LIN {X 0,Y 383.012,Z 410.276,A -85,B 0,C 180,E1 -11840.414,E2 -11840.414} C_VEL
LIN {X 0,Y 383.022,Z 410.276,A -85,B 0,C 180,E1 -11844.045,E2 -11844.045} C_VEL
LIN {X 0,Y 383.032,Z 410.273,A -85,B 0,C 180,E1 -11847.853,E2 -11847.853} C_VEL
LIN {X 0,Y 383.059,Z 410.269,A -85,B 0,C 180,E1 -11851.721,E2 -11851.721} C_VEL
LIN {X 0,Y 383.047,Z 410.267,A -85,B 0,C 180,E1 -11855.04,E2 -11855.04} C_VEL
LIN {X 0,Y 382.989,Z 410.276,A -85,B 0,C 180,E1 -11858.469,E2 -11858.469} C_VEL
LIN {X 0,Y 383.085,Z 410.269,A -85,B 0,C 180,E1 -11861.828,E2 -11861.828} C_VEL
LIN {X 0,Y 383.108,Z 410.26,A -85,B 0,C 180,E1 -11865.119,E2 -11865.119} C_VEL
LIN {X 0,Y 383.093,Z 410.263,A -85,B 0,C 180,E1 -11868.358,E2 -11868.358} C_VEL
LIN {X 0,Y 383.3,Z 410.24,A -85,B 0,C 180,E1 -11871.934,E2 -11871.934} C_VEL
LIN {X 0,Y 383.196,Z 410.249,A -85,B 0,C 180,E1 -11874.739,E2 -11874.739} C_VEL
LIN {X 0,Y 383.384,Z 410.229,A -85,B 0,C 180,E1 -11877.899,E2 -11877.899} C_VEL
LIN {X 0,Y 383.516,Z 410.211,A -85,B 0,C 180,E1 -11880.001,E2 -11880.001} C_VEL
LIN {X 0,Y 383.249,Z 410.245,A -85,B 0,C 180,E1 -11883.154,E2 -11883.154} C_VEL
LIN {X 0,Y 383.284,Z 410.238,A -85,B 0,C 180,E1 -11886.317,E2 -11886.317} C_VEL
LIN {X 0,Y 383.257,Z 410.241,A -85,B 0,C 180,E1 -11888.436,E2 -11888.436} C_VEL
LIN {X 0,Y 383.095,Z 410.266,A -85,B 0,C 180,E1 -11891.643,E2 -11891.643} C_VEL
LIN {X 0,Y 383.108,Z 410.261,A -85,B 0,C 180,E1 -11894.882,E2 -11894.882} C_VEL
LIN {X 0,Y 383.061,Z 410.266,A -85,B 0,C 180,E1 -11898.174,E2 -11898.174} C_VEL
LIN {X 0,Y 382.991,Z 410.278,A -85,B 0,C 180,E1 -11901.532,E2 -11901.532} C_VEL
LIN {X 0,Y 383.051,Z 410.271,A -85,B 0,C 180,E1 -11904.961,E2 -11904.961} C_VEL
LIN {X 0,Y 383.028,Z 410.27,A -85,B 0,C 180,E1 -11908.271,E2 -11908.271} C_VEL
LIN {X 0,Y 383.008,Z 410.272,A -85,B 0,C 180,E1 -11912.15,E2 -11912.15} C_VEL
LIN {X 0,Y 383.018,Z 410.274,A -85,B 0,C 180,E1 -11914.669,E2 -11914.669} C_VEL
LIN {X 0,Y 383.004,Z 410.278,A -85,B 0,C 180,E1 -11917.905,E2 -11917.905} C_VEL
LIN {X 0,Y 383.441,Z 413.021,A -85,B 0,C 180,E1 -11921.288,E2 -11921.288} C_VEL
LIN {X 0,Y 383.863,Z 416.004,A -85,B 0,C 180,E1 -11924.436,E2 -11924.436} C_VEL
LIN {X 0,Y 384.216,Z 419.062,A -85,B 0,C 180,E1 -11927.407,E2 -11927.407} C_VEL
LIN {X 0,Y 384.099,Z 422.233,A -85,B 0,C 180,E1 -11930.219,E2 -11930.219} C_VEL
LIN {X 0,Y 383.629,Z 426.471,A -85,B 0,C 180,E1 -11933.714,E2 -11933.714} C_VEL
LIN {X 0,Y 383.227,Z 430.206,A -85,B 0,C 180,E1 -11936.622,E2 -11936.622} C_VEL
LIN {X 0,Y 382.802,Z 435.145,A -85,B 0,C 180,E1 -11940.284,E2 -11940.284} C_VEL
LIN {X 0,Y 382.563,Z 438.484,A -85,B 0,C 180,E1 -11942.66,E2 -11942.66} C_VEL
LIN {X 0,Y 382.356,Z 441.851,A -85,B 0,C 180,E1 -11944.991,E2 -11944.991} C_VEL
LIN {X 0,Y 382.084,Z 446.961,A -85,B 0,C 180,E1 -11948.415,E2 -11948.415} C_VEL
LIN {X 0,Y 381.915,Z 451.227,A -85,B 0,C 180,E1 -11951.101,E2 -11951.101} C_VEL
LIN {X 0,Y 383.99,Z 461.506,A -85,B 0,C 180,E1 -11951.544,E2 -11951.544} C_VEL
LIN {X 0,Y 385.644,Z 470.976,A -85,B 0,C 180,E1 -11952.061,E2 -11952.061} C_VEL
LIN {X 0,Y 386.955,Z 479.684,A -85,B 0,C 180,E1 -11952.632,E2 -11952.632} C_VEL
LIN {X 0,Y 387.304,Z 485.306,A -85,B 0,C 180,E1 -11953.027,E2 -11953.027} C_VEL
LIN {X 0,Y 386.288,Z 497.459,A -85,B 0,C 180,E1 -11954.027,E2 -11954.027} C_VEL
LIN {X 0,Y 385.499,Z 506.412,A -85,B 0,C 180,E1 -11954.943,E2 -11954.943} C_VEL
LIN {X 0,Y 384.91,Z 513.425,A -85,B 0,C 180,E1 -11955.786,E2 -11955.786} C_VEL
LIN {X 0,Y 384.102,Z 522.165,A -85,B 0,C 180,E1 -11957.048,E2 -11957.048} C_VEL
LIN {X 0,Y 383.437,Z 528.368,A -85,B 0,C 180,E1 -11958.1,E2 -11958.1} C_VEL
LIN {X 0,Y 382.892,Z 534.91,A -85,B 0,C 180,E1 -11959.423,E2 -11959.423} C_VEL
LIN {X 0,Y 382.464,Z 539.413,A -85,B 0,C 180,E1 -11960.481,E2 -11960.481} C_VEL
LIN {X 0,Y 382.033,Z 544.907,A -85,B 0,C 180,E1 -11962.069,E2 -11962.069} C_VEL
LIN {X 0,Y 381.769,Z 549.234,A -85,B 0,C 180,E1 -11963.658,E2 -11963.658} C_VEL
LIN {X 0,Y 381.682,Z 551.602,A -85,B 0,C 180,E1 -11964.717,E2 -11964.717} C_VEL
LIN {X 0,Y 381.642,Z 553.402,A -85,B 0,C 180,E1 -11965.776,E2 -11965.776} C_VEL
LIN {X 0,Y 381.558,Z 555.847,A -85,B 0,C 180,E1 -11967.889,E2 -11967.889} C_VEL
LIN {X 0,Y 381.591,Z 556.437,A -85,B 0,C 180,E1 -11968.944,E2 -11968.944} C_VEL
LIN {X 0,Y 381.591,Z 556.437,A -85,B 0,C 180,E1 -11971.055,E2 -11971.055} C_VEL
LIN {X 0,Y 381.558,Z 555.848,A -85,B 0,C 180,E1 -11972.111,E2 -11972.111} C_VEL
LIN {X 0,Y 381.642,Z 553.403,A -85,B 0,C 180,E1 -11974.224,E2 -11974.224} C_VEL
LIN {X 0,Y 381.693,Z 550.488,A -85,B 0,C 180,E1 -11975.796,E2 -11975.796} C_VEL
LIN {X 0,Y 381.934,Z 546.463,A -85,B 0,C 180,E1 -11977.4,E2 -11977.4} C_VEL
LIN {X 0,Y 382.305,Z 541.331,A -85,B 0,C 180,E1 -11978.989,E2 -11978.989} C_VEL
LIN {X 0,Y 382.759,Z 536.068,A -85,B 0,C 180,E1 -11980.313,E2 -11980.313} C_VEL
LIN {X 0,Y 383.293,Z 529.747,A -85,B 0,C 180,E1 -11981.636,E2 -11981.636} C_VEL
LIN {X 0,Y 383.909,Z 523.795,A -85,B 0,C 180,E1 -11982.69,E2 -11982.69} C_VEL
LIN {X 0,Y 384.57,Z 516.865,A -85,B 0,C 180,E1 -11983.743,E2 -11983.743} C_VEL
LIN {X 0,Y 385.262,Z 508.68,A -85,B 0,C 180,E1 -11984.796,E2 -11984.796} C_VEL
LIN {X 0,Y 386.03,Z 500.167,A -85,B 0,C 180,E1 -11985.712,E2 -11985.712} C_VEL
LIN {X 0,Y 386.744,Z 491.448,A -85,B 0,C 180,E1 -11986.495,E2 -11986.495} C_VEL
LIN {X 0,Y 387.323,Z 482.508,A -85,B 0,C 180,E1 -11987.161,E2 -11987.161} C_VEL
LIN {X 0,Y 385.932,Z 472.449,A -85,B 0,C 180,E1 -11987.848,E2 -11987.848} C_VEL
LIN {X 0,Y 384.09,Z 461.865,A -85,B 0,C 180,E1 -11988.437,E2 -11988.437} C_VEL
LIN {X 0,Y 381.971,Z 451.872,A -85,B 0,C 180,E1 -11988.879,E2 -11988.879} C_VEL
LIN {X 0,Y 381.884,Z 451.048,A -85,B 0,C 180,E1 -11988.926,E2 -11988.926} C_VEL
LIN {X 0,Y 382.184,Z 445.234,A -85,B 0,C 180,E1 -11992.716,E2 -11992.716} C_VEL
LIN {X 0,Y 382.45,Z 440.161,A -85,B 0,C 180,E1 -11996.169,E2 -11996.169} C_VEL
LIN {X 0,Y 382.796,Z 435.146,A -85,B 0,C 180,E1 -11999.716,E2 -11999.716} C_VEL
LIN {X 0,Y 383.224,Z 430.206,A -85,B 0,C 180,E1 -12003.378,E2 -12003.378} C_VEL
LIN {X 0,Y 383.748,Z 425.351,A -85,B 0,C 180,E1 -12007.182,E2 -12007.182} C_VEL
LIN {X 0,Y 384.098,Z 422.187,A -85,B 0,C 180,E1 -12009.821,E2 -12009.821} C_VEL
LIN {X 0,Y 384.212,Z 419.044,A -85,B 0,C 180,E1 -12012.593,E2 -12012.593} C_VEL
LIN {X 0,Y 383.827,Z 415.64,A -85,B 0,C 180,E1 -12015.909,E2 -12015.909} C_VEL
LIN {X 0,Y 383.416,Z 412.995,A -85,B 0,C 180,E1 -12018.722,E2 -12018.722} C_VEL
LIN {X 0,Y 383.001,Z 410.279,A -85,B 0,C 180,E1 -12022.095,E2 -12022.095} C_VEL
LIN {X 0,Y 383.015,Z 410.277,A -85,B 0,C 180,E1 -12025.331,E2 -12025.331} C_VEL
LIN {X 0,Y 383.034,Z 410.269,A -85,B 0,C 180,E1 -12027.852,E2 -12027.852} C_VEL
LIN {X 0,Y 383.06,Z 410.266,A -85,B 0,C 180,E1 -12031.719,E2 -12031.719} C_VEL
LIN {X 0,Y 383.048,Z 410.271,A -85,B 0,C 180,E1 -12035.039,E2 -12035.039} C_VEL
LIN {X 0,Y 382.988,Z 410.278,A -85,B 0,C 180,E1 -12038.468,E2 -12038.468} C_VEL
LIN {X 0,Y 383.058,Z 410.266,A -85,B 0,C 180,E1 -12041.826,E2 -12041.826} C_VEL
LIN {X 0,Y 383.105,Z 410.262,A -85,B 0,C 180,E1 -12045.118,E2 -12045.118} C_VEL
LIN {X 0,Y 383.093,Z 410.266,A -85,B 0,C 180,E1 -12048.357,E2 -12048.357} C_VEL
LIN {X 0,Y 383.298,Z 410.237,A -85,B 0,C 180,E1 -12051.932,E2 -12051.932} C_VEL
LIN {X 0,Y 383.194,Z 410.253,A -85,B 0,C 180,E1 -12054.738,E2 -12054.738} C_VEL
LIN {X 0,Y 383.382,Z 410.227,A -85,B 0,C 180,E1 -12057.898,E2 -12057.898} C_VEL
LIN {X 0,Y 383.513,Z 410.212,A -85,B 0,C 180,E1 -12059.999,E2 -12059.999} C_VEL
LIN {X 0,Y 383.246,Z 410.243,A -85,B 0,C 180,E1 -12063.153,E2 -12063.153} C_VEL
LIN {X 0,Y 383.262,Z 410.243,A -85,B 0,C 180,E1 -12066.636,E2 -12066.636} C_VEL
LIN {X 0,Y 383.253,Z 410.246,A -85,B 0,C 180,E1 -12068.435,E2 -12068.435} C_VEL
LIN {X 0,Y 383.09,Z 410.263,A -85,B 0,C 180,E1 -12071.642,E2 -12071.642} C_VEL
LIN {X 0,Y 383.106,Z 410.26,A -85,B 0,C 180,E1 -12074.881,E2 -12074.881} C_VEL
LIN {X 0,Y 383.082,Z 410.269,A -85,B 0,C 180,E1 -12078.172,E2 -12078.172} C_VEL
LIN {X 0,Y 382.986,Z 410.276,A -85,B 0,C 180,E1 -12081.531,E2 -12081.531} C_VEL
LIN {X 0,Y 383.045,Z 410.267,A -85,B 0,C 180,E1 -12084.96,E2 -12084.96} C_VEL
LIN {X 0,Y 383.042,Z 410.269,A -85,B 0,C 180,E1 -12088.492,E2 -12088.492} C_VEL
LIN {X 0,Y 383.001,Z 410.274,A -85,B 0,C 180,E1 -12092.427,E2 -12092.427} C_VEL
LIN {X 0,Y 383.027,Z 410.273,A -85,B 0,C 180,E1 -12096.165,E2 -12096.165} C_VEL
LIN {X 0,Y 383.014,Z 410.276,A -85,B 0,C 180,E1 -12099.957,E2 -12099.957} C_VEL
LIN {X 0,Y 383.059,Z 410.266,A -85,B 0,C 180,E1 -12102.788,E2 -12102.788} C_VEL
LIN {X 0,Y 383.063,Z 410.271,A -85,B 0,C 180,E1 -12105.8,E2 -12105.8} C_VEL
LIN {X 0,Y 383.038,Z 410.269,A -85,B 0,C 180,E1 -12108.786,E2 -12108.786} C_VEL
LIN {X 0,Y 382.997,Z 410.275,A -85,B 0,C 180,E1 -12112.096,E2 -12112.096} C_VEL
LIN {X 0,Y 383.012,Z 410.276,A -85,B 0,C 180,E1 -12115.332,E2 -12115.332} C_VEL
LIN {X 0,Y 382.977,Z 410.278,A -85,B 0,C 180,E1 -12119.082,E2 -12119.082} C_VEL
LIN {X 0,Y 383.051,Z 410.267,A -85,B 0,C 180,E1 -12122.698,E2 -12122.698} C_VEL
LIN {X 0,Y 383.029,Z 410.27,A -85,B 0,C 180,E1 -12126.193,E2 -12126.193} C_VEL
LIN {X 0,Y 383.05,Z 410.272,A -85,B 0,C 180,E1 -12129.599,E2 -12129.599} C_VEL
LIN {X 0,Y 383.1,Z 410.267,A -85,B 0,C 180,E1 -12132.932,E2 -12132.932} C_VEL
LIN {X 0,Y 383.121,Z 410.263,A -85,B 0,C 180,E1 -12136.464,E2 -12136.464} C_VEL
LIN {X 0,Y 383.138,Z 410.29,A -85,B 0,C 180,E1 -12139.598,E2 -12139.598} C_VEL
LIN {X 0,Y 383.821,Z 412.514,A -85,B 0,C 180,E1 -12139.95,E2 -12139.95} C_VEL
LIN {X 0,Y 385.2,Z 414.425,A -85,B 0,C 180,E1 -12140.616,E2 -12140.616} C_VEL
LIN {X 0,Y 387.436,Z 415.861,A -85,B 0,C 180,E1 -12141.656,E2 -12141.656} C_VEL
LIN {X 0,Y 388.84,Z 416.571,A -85,B 0,C 180,E1 -12142.402,E2 -12142.402} C_VEL
LIN {X 0,Y 389.961,Z 418.835,A -85,B 0,C 180,E1 -12143.142,E2 -12143.142} C_VEL
LIN {X 0,Y 391.789,Z 420.996,A -85,B 0,C 180,E1 -12144.467,E2 -12144.467} C_VEL
LIN {X 0,Y 393.422,Z 422.061,A -85,B 0,C 180,E1 -12145.903,E2 -12145.903} C_VEL
LIN {X 0,Y 394.945,Z 422.431,A -85,B 0,C 180,E1 -12147.961,E2 -12147.961} C_VEL
LIN {X 0,Y 395.509,Z 422.495,A -85,B 0,C 180,E1 -12150,E2 -12150} C_VEL
LIN {X 0,Y 394.944,Z 422.431,A -85,B 0,C 180,E1 -12152.04,E2 -12152.04} C_VEL
LIN {X 0,Y 393.422,Z 422.061,A -85,B 0,C 180,E1 -12154.098,E2 -12154.098} C_VEL
LIN {X 0,Y 391.445,Z 420.7,A -85,B 0,C 180,E1 -12155.796,E2 -12155.796} C_VEL
LIN {X 0,Y 389.551,Z 418.154,A -85,B 0,C 180,E1 -12157.135,E2 -12157.135} C_VEL
LIN {X 0,Y 388.788,Z 416.393,A -85,B 0,C 180,E1 -12157.634,E2 -12157.634} C_VEL
LIN {X 0,Y 385.957,Z 415.054,A -85,B 0,C 180,E1 -12159.036,E2 -12159.036} C_VEL
LIN {X 0,Y 384.054,Z 412.961,A -85,B 0,C 180,E1 -12159.938,E2 -12159.938} C_VEL
LIN {X 0,Y 383.253,Z 410.919,A -85,B 0,C 180,E1 -12160.333,E2 -12160.333} C_VEL
LIN {X 0,Y 383.122,Z 410.263,A -85,B 0,C 180,E1 -12160.437,E2 -12160.437} C_VEL
LIN {X 0,Y 383.123,Z 410.262,A -85,B 0,C 180,E1 -12163.796,E2 -12163.796} C_VEL
LIN {X 0,Y 383.091,Z 410.267,A -85,B 0,C 180,E1 -12167.455,E2 -12167.455} C_VEL
LIN {X 0,Y 383.025,Z 410.276,A -85,B 0,C 180,E1 -12170.647,E2 -12170.647} C_VEL
LIN {X 0,Y 383.03,Z 410.27,A -85,B 0,C 180,E1 -12173.807,E2 -12173.807} C_VEL
LIN {X 0,Y 383.053,Z 410.267,A -85,B 0,C 180,E1 -12177.302,E2 -12177.302} C_VEL
LIN {X 0,Y 382.978,Z 410.278,A -85,B 0,C 180,E1 -12180.919,E2 -12180.919} C_VEL
LIN {X 0,Y 383.014,Z 410.276,A -85,B 0,C 180,E1 -12184.668,E2 -12184.668} C_VEL
LIN {X 0,Y 382.995,Z 410.274,A -85,B 0,C 180,E1 -12185.381,E2 -12185.381} C_VEL
LIN {X 0,Y 382.352,Z 410.358,A -85,B 0,C 180,E1 -12186.258,E2 -12186.258} C_VEL
LIN {X 0,Y 379.535,Z 410.71,A -85,B 0,C 180,E1 -12187.686,E2 -12187.686} C_VEL
LIN {X 0,Y 377.13,Z 411.01,A -85,B 0,C 180,E1 -12188.841,E2 -12188.841} C_VEL
LIN {X 0,Y 376.084,Z 411.138,A -85,B 0,C 180,E1 -12189.733,E2 -12189.733} C_VEL
LIN {X 0,Y 375.992,Z 411.148,A -85,B 0,C 180,E1 -12190.035,E2 -12190.035} C_VEL
LIN {X 0,Y 375.984,Z 411.147,A -85,B 0,C 180,E1 -12193.198,E2 -12193.198} C_VEL
LIN {X 0,Y 375.932,Z 411.155,A -85,B 0,C 180,E1 -12196.81,E2 -12196.81} C_VEL
LIN {X 0,Y 375.959,Z 411.153,A -85,B 0,C 180,E1 -12200.538,E2 -12200.538} C_VEL
LIN {X 0,Y 375.96,Z 411.151,A -85,B 0,C 180,E1 -12203.496,E2 -12203.496} C_VEL
LIN {X 0,Y 375.959,Z 411.154,A -85,B 0,C 180,E1 -12205.889,E2 -12205.889} C_VEL
LIN {X 0,Y 375.965,Z 411.152,A -85,B 0,C 180,E1 -12209.688,E2 -12209.688} C_VEL
LIN {X 0,Y 375.998,Z 411.151,A -85,B 0,C 180,E1 -12212.142,E2 -12212.142} C_VEL
LIN {X 0,Y 376.001,Z 411.146,A -85,B 0,C 180,E1 -12214.539,E2 -12214.539} C_VEL
LIN {X 0,Y 375.959,Z 411.156,A -85,B 0,C 180,E1 -12218.046,E2 -12218.046} C_VEL
LIN {X 0,Y 376.02,Z 411.145,A -85,B 0,C 180,E1 -12221.474,E2 -12221.474} C_VEL
LIN {X 0,Y 376.057,Z 411.138,A -85,B 0,C 180,E1 -12224.833,E2 -12224.833} C_VEL
LIN {X 0,Y 376.046,Z 411.142,A -85,B 0,C 180,E1 -12228.137,E2 -12228.137} C_VEL
LIN {X 0,Y 376.254,Z 411.119,A -85,B 0,C 180,E1 -12231.878,E2 -12231.878} C_VEL
LIN {X 0,Y 376.168,Z 411.124,A -85,B 0,C 180,E1 -12234.64,E2 -12234.64} C_VEL
LIN {X 0,Y 376.35,Z 411.106,A -85,B 0,C 180,E1 -12237.86,E2 -12237.86} C_VEL
LIN {X 0,Y 376.485,Z 411.087,A -85,B 0,C 180,E1 -12240.001,E2 -12240.001} C_VEL
LIN {X 0,Y 376.187,Z 411.125,A -85,B 0,C 180,E1 -12243.214,E2 -12243.214} C_VEL
LIN {X 0,Y 376.244,Z 411.115,A -85,B 0,C 180,E1 -12246.436,E2 -12246.436} C_VEL
LIN {X 0,Y 376.203,Z 411.12,A -85,B 0,C 180,E1 -12248.596,E2 -12248.596} C_VEL
LIN {X 0,Y 376.048,Z 411.141,A -85,B 0,C 180,E1 -12251.864,E2 -12251.864} C_VEL
LIN {X 0,Y 376.056,Z 411.142,A -85,B 0,C 180,E1 -12255.168,E2 -12255.168} C_VEL
LIN {X 0,Y 376.007,Z 411.144,A -85,B 0,C 180,E1 -12258.527,E2 -12258.527} C_VEL
LIN {X 0,Y 375.961,Z 411.151,A -85,B 0,C 180,E1 -12261.955,E2 -12261.955} C_VEL
LIN {X 0,Y 376.005,Z 411.148,A -85,B 0,C 180,E1 -12265.462,E2 -12265.462} C_VEL
LIN {X 0,Y 375.96,Z 411.156,A -85,B 0,C 180,E1 -12269.081,E2 -12269.081} C_VEL
LIN {X 0,Y 375.948,Z 411.155,A -85,B 0,C 180,E1 -12272.829,E2 -12272.829} C_VEL
LIN {X 0,Y 375.958,Z 411.157,A -85,B 0,C 180,E1 -12275.416,E2 -12275.416} C_VEL
LIN {X 0,Y 375.994,Z 411.434,A -85,B 0,C 180,E1 -12278.086,E2 -12278.086} C_VEL
LIN {X 0,Y 376.472,Z 414.514,A -85,B 0,C 180,E1 -12281.693,E2 -12281.693} C_VEL
LIN {X 0,Y 376.939,Z 417.754,A -85,B 0,C 180,E1 -12285.114,E2 -12285.114} C_VEL
LIN {X 0,Y 377.173,Z 420.932,A -85,B 0,C 180,E1 -12288.189,E2 -12288.189} C_VEL
LIN {X 0,Y 376.989,Z 423.718,A -85,B 0,C 180,E1 -12290.666,E2 -12290.666} C_VEL
LIN {X 0,Y 376.633,Z 426.928,A -85,B 0,C 180,E1 -12293.359,E2 -12293.359} C_VEL
LIN {X 0,Y 376.255,Z 430.124,A -85,B 0,C 180,E1 -12295.919,E2 -12295.919} C_VEL
LIN {X 0,Y 375.826,Z 435.042,A -85,B 0,C 180,E1 -12299.675,E2 -12299.675} C_VEL
LIN {X 0,Y 375.558,Z 438.367,A -85,B 0,C 180,E1 -12302.106,E2 -12302.106} C_VEL
LIN {X 0,Y 375.358,Z 441.711,A -85,B 0,C 180,E1 -12304.492,E2 -12304.492} C_VEL
LIN {X 0,Y 375.018,Z 446.771,A -85,B 0,C 180,E1 -12307.988,E2 -12307.988} C_VEL
LIN {X 0,Y 374.845,Z 450.829,A -85,B 0,C 180,E1 -12310.704,E2 -12310.704} C_VEL
LIN {X 0,Y 377.83,Z 465.657,A -85,B 0,C 180,E1 -12311.408,E2 -12311.408} C_VEL
LIN {X 0,Y 379.809,Z 478.486,A -85,B 0,C 180,E1 -12312.228,E2 -12312.228} C_VEL
LIN {X 0,Y 380.475,Z 485.161,A -85,B 0,C 180,E1 -12312.718,E2 -12312.718} C_VEL
LIN {X 0,Y 379.452,Z 497.247,A -85,B 0,C 180,E1 -12313.732,E2 -12313.732} C_VEL
LIN {X 0,Y 378.606,Z 506.195,A -85,B 0,C 180,E1 -12314.662,E2 -12314.662} C_VEL
LIN {X 0,Y 377.976,Z 513.549,A -85,B 0,C 180,E1 -12315.568,E2 -12315.568} C_VEL
LIN {X 0,Y 377.173,Z 521.954,A -85,B 0,C 180,E1 -12316.805,E2 -12316.805} C_VEL
LIN {X 0,Y 376.471,Z 528.156,A -85,B 0,C 180,E1 -12317.877,E2 -12317.877} C_VEL
LIN {X 0,Y 375.857,Z 534.697,A -85,B 0,C 180,E1 -12319.223,E2 -12319.223} C_VEL
LIN {X 0,Y 375.45,Z 539.201,A -85,B 0,C 180,E1 -12320.301,E2 -12320.301} C_VEL
LIN {X 0,Y 374.964,Z 544.695,A -85,B 0,C 180,E1 -12321.919,E2 -12321.919} C_VEL
LIN {X 0,Y 374.685,Z 549.022,A -85,B 0,C 180,E1 -12323.538,E2 -12323.538} C_VEL
LIN {X 0,Y 374.588,Z 551.39,A -85,B 0,C 180,E1 -12324.617,E2 -12324.617} C_VEL
LIN {X 0,Y 374.569,Z 553.191,A -85,B 0,C 180,E1 -12325.696,E2 -12325.696} C_VEL
LIN {X 0,Y 374.457,Z 555.636,A -85,B 0,C 180,E1 -12327.849,E2 -12327.849} C_VEL
LIN {X 0,Y 374.492,Z 556.226,A -85,B 0,C 180,E1 -12328.924,E2 -12328.924} C_VEL
LIN {X 0,Y 374.492,Z 556.226,A -85,B 0,C 180,E1 -12331.075,E2 -12331.075} C_VEL
LIN {X 0,Y 374.457,Z 555.636,A -85,B 0,C 180,E1 -12332.151,E2 -12332.151} C_VEL
LIN {X 0,Y 374.569,Z 553.192,A -85,B 0,C 180,E1 -12334.304,E2 -12334.304} C_VEL
LIN {X 0,Y 374.591,Z 551.391,A -85,B 0,C 180,E1 -12335.382,E2 -12335.382} C_VEL
LIN {X 0,Y 374.77,Z 547.782,A -85,B 0,C 180,E1 -12337.001,E2 -12337.001} C_VEL
LIN {X 0,Y 375.102,Z 543.035,A -85,B 0,C 180,E1 -12338.62,E2 -12338.62} C_VEL
LIN {X 0,Y 375.628,Z 537.011,A -85,B 0,C 180,E1 -12340.238,E2 -12340.238} C_VEL
LIN {X 0,Y 376.189,Z 530.911,A -85,B 0,C 180,E1 -12341.585,E2 -12341.585} C_VEL
LIN {X 0,Y 376.975,Z 523.583,A -85,B 0,C 180,E1 -12342.927,E2 -12342.927} C_VEL
LIN {X 0,Y 377.631,Z 516.653,A -85,B 0,C 180,E1 -12344.001,E2 -12344.001} C_VEL
LIN {X 0,Y 378.389,Z 508.469,A -85,B 0,C 180,E1 -12345.071,E2 -12345.071} C_VEL
LIN {X 0,Y 379.168,Z 499.955,A -85,B 0,C 180,E1 -12346.004,E2 -12346.004} C_VEL
LIN {X 0,Y 379.95,Z 491.237,A -85,B 0,C 180,E1 -12346.799,E2 -12346.799} C_VEL
LIN {X 0,Y 380.478,Z 483.846,A -85,B 0,C 180,E1 -12347.373,E2 -12347.373} C_VEL
LIN {X 0,Y 378.98,Z 472.564,A -85,B 0,C 180,E1 -12348.168,E2 -12348.168} C_VEL
LIN {X 0,Y 377.134,Z 462.285,A -85,B 0,C 180,E1 -12348.764,E2 -12348.764} C_VEL
LIN {X 0,Y 374.921,Z 451.691,A -85,B 0,C 180,E1 -12349.247,E2 -12349.247} C_VEL
LIN {X 0,Y 374.844,Z 450.829,A -85,B 0,C 180,E1 -12349.295,E2 -12349.295} C_VEL
LIN {X 0,Y 375.14,Z 444.785,A -85,B 0,C 180,E1 -12353.366,E2 -12353.366} C_VEL
LIN {X 0,Y 375.403,Z 440.027,A -85,B 0,C 180,E1 -12356.699,E2 -12356.699} C_VEL
LIN {X 0,Y 375.823,Z 435.042,A -85,B 0,C 180,E1 -12360.324,E2 -12360.324} C_VEL
LIN {X 0,Y 376.253,Z 430.125,A -85,B 0,C 180,E1 -12364.08,E2 -12364.08} C_VEL
LIN {X 0,Y 376.634,Z 426.901,A -85,B 0,C 180,E1 -12366.663,E2 -12366.663} C_VEL
LIN {X 0,Y 377.085,Z 422.756,A -85,B 0,C 180,E1 -12370.168,E2 -12370.168} C_VEL
LIN {X 0,Y 377.165,Z 420.57,A -85,B 0,C 180,E1 -12372.129,E2 -12372.129} C_VEL
LIN {X 0,Y 376.914,Z 417.497,A -85,B 0,C 180,E1 -12375.116,E2 -12375.116} C_VEL
LIN {X 0,Y 376.453,Z 414.513,A -85,B 0,C 180,E1 -12378.309,E2 -12378.309} C_VEL
LIN {X 0,Y 375.992,Z 411.438,A -85,B 0,C 180,E1 -12381.914,E2 -12381.914} C_VEL
LIN {X 0,Y 375.955,Z 411.156,A -85,B 0,C 180,E1 -12384.584,E2 -12384.584} C_VEL
LIN {X 0,Y 375.974,Z 411.15,A -85,B 0,C 180,E1 -12388.439,E2 -12388.439} C_VEL
LIN {X 0,Y 375.999,Z 411.146,A -85,B 0,C 180,E1 -12392.141,E2 -12392.141} C_VEL
LIN {X 0,Y 376.002,Z 411.149,A -85,B 0,C 180,E1 -12394.538,E2 -12394.538} C_VEL
LIN {X 0,Y 375.958,Z 411.151,A -85,B 0,C 180,E1 -12398.045,E2 -12398.045} C_VEL
LIN {X 0,Y 376.004,Z 411.145,A -85,B 0,C 180,E1 -12401.472,E2 -12401.472} C_VEL
LIN {X 0,Y 376.053,Z 411.143,A -85,B 0,C 180,E1 -12404.832,E2 -12404.832} C_VEL
LIN {X 0,Y 376.045,Z 411.142,A -85,B 0,C 180,E1 -12408.136,E2 -12408.136} C_VEL
LIN {X 0,Y 376.252,Z 411.115,A -85,B 0,C 180,E1 -12411.877,E2 -12411.877} C_VEL
LIN {X 0,Y 376.166,Z 411.129,A -85,B 0,C 180,E1 -12414.639,E2 -12414.639} C_VEL
LIN {X 0,Y 376.348,Z 411.103,A -85,B 0,C 180,E1 -12417.859,E2 -12417.859} C_VEL
LIN {X 0,Y 376.483,Z 411.088,A -85,B 0,C 180,E1 -12419.999,E2 -12419.999} C_VEL
LIN {X 0,Y 376.184,Z 411.122,A -85,B 0,C 180,E1 -12423.212,E2 -12423.212} C_VEL
LIN {X 0,Y 376.227,Z 411.12,A -85,B 0,C 180,E1 -12426.627,E2 -12426.627} C_VEL
LIN {X 0,Y 376.199,Z 411.123,A -85,B 0,C 180,E1 -12428.595,E2 -12428.595} C_VEL
LIN {X 0,Y 376.043,Z 411.143,A -85,B 0,C 180,E1 -12431.863,E2 -12431.863} C_VEL
LIN {X 0,Y 376.054,Z 411.138,A -85,B 0,C 180,E1 -12435.167,E2 -12435.167} C_VEL
LIN {X 0,Y 376.017,Z 411.145,A -85,B 0,C 180,E1 -12438.526,E2 -12438.526} C_VEL
LIN {X 0,Y 375.956,Z 411.156,A -85,B 0,C 180,E1 -12441.954,E2 -12441.954} C_VEL
LIN {X 0,Y 375.999,Z 411.147,A -85,B 0,C 180,E1 -12445.461,E2 -12445.461} C_VEL
LIN {X 0,Y 375.97,Z 411.149,A -85,B 0,C 180,E1 -12449.078,E2 -12449.078} C_VEL
LIN {X 0,Y 375.951,Z 411.151,A -85,B 0,C 180,E1 -12452.828,E2 -12452.828} C_VEL
LIN {X 0,Y 375.951,Z 411.153,A -85,B 0,C 180,E1 -12455.415,E2 -12455.415} C_VEL
LIN {X 0,Y 375.971,Z 411.151,A -85,B 0,C 180,E1 -12458.271,E2 -12458.271} C_VEL
LIN {X 0,Y 375.983,Z 411.152,A -85,B 0,C 180,E1 -12461.61,E2 -12461.61} C_VEL
LIN {X 0,Y 376.009,Z 411.146,A -85,B 0,C 180,E1 -12465.255,E2 -12465.255} C_VEL
LIN {X 0,Y 375.983,Z 411.148,A -85,B 0,C 180,E1 -12468.39,E2 -12468.39} C_VEL
LIN {X 0,Y 375.962,Z 411.153,A -85,B 0,C 180,E1 -12471.912,E2 -12471.912} C_VEL
LIN {X 0,Y 375.974,Z 411.153,A -85,B 0,C 180,E1 -12475.333,E2 -12475.333} C_VEL
LIN {X 0,Y 375.952,Z 411.151,A -85,B 0,C 180,E1 -12478.438,E2 -12478.438} C_VEL
LIN {X 0,Y 375.99,Z 411.147,A -85,B 0,C 180,E1 -12482.142,E2 -12482.142} C_VEL
LIN {X 0,Y 376.001,Z 411.145,A -85,B 0,C 180,E1 -12484.539,E2 -12484.539} C_VEL
LIN {X 0,Y 375.958,Z 411.151,A -85,B 0,C 180,E1 -12488.046,E2 -12488.046} C_VEL
LIN {X 0,Y 376.019,Z 411.148,A -85,B 0,C 180,E1 -12491.474,E2 -12491.474} C_VEL
LIN {X 0,Y 376.054,Z 411.144,A -85,B 0,C 180,E1 -12494.833,E2 -12494.833} C_VEL
LIN {X 0,Y 376.117,Z 411.323,A -85,B 0,C 180,E1 -12497.317,E2 -12497.317} C_VEL
LIN {X 0,Y 376.774,Z 413.474,A -85,B 0,C 180,E1 -12497.614,E2 -12497.614} C_VEL
LIN {X 0,Y 378.392,Z 415.585,A -85,B 0,C 180,E1 -12498.211,E2 -12498.211} C_VEL
LIN {X 0,Y 380.855,Z 416.996,A -85,B 0,C 180,E1 -12499.097,E2 -12499.097} C_VEL
LIN {X 0,Y 381.348,Z 417.795,A -85,B 0,C 180,E1 -12499.313,E2 -12499.313} C_VEL
LIN {X 0,Y 382.988,Z 420.389,A -85,B 0,C 180,E1 -12500.027,E2 -12500.027} C_VEL
LIN {X 0,Y 385.3,Z 422.351,A -85,B 0,C 180,E1 -12501.081,E2 -12501.081} C_VEL
LIN {X 0,Y 387.405,Z 423.442,A -85,B 0,C 180,E1 -12502.125,E2 -12502.125} C_VEL
LIN {X 0,Y 388.935,Z 426,A -85,B 0,C 180,E1 -12503.079,E2 -12503.079} C_VEL
LIN {X 0,Y 390.889,Z 428.078,A -85,B 0,C 180,E1 -12504.455,E2 -12504.455} C_VEL
LIN {X 0,Y 392.534,Z 429.095,A -85,B 0,C 180,E1 -12505.893,E2 -12505.893} C_VEL
LIN {X 0,Y 394.082,Z 429.478,A -85,B 0,C 180,E1 -12507.956,E2 -12507.956} C_VEL
LIN {X 0,Y 394.645,Z 429.534,A -85,B 0,C 180,E1 -12510,E2 -12510} C_VEL
LIN {X 0,Y 394.082,Z 429.477,A -85,B 0,C 180,E1 -12512.044,E2 -12512.044} C_VEL
LIN {X 0,Y 392.534,Z 429.092,A -85,B 0,C 180,E1 -12514.107,E2 -12514.107} C_VEL
LIN {X 0,Y 390.529,Z 427.797,A -85,B 0,C 180,E1 -12515.81,E2 -12515.81} C_VEL
LIN {X 0,Y 388.493,Z 425.353,A -85,B 0,C 180,E1 -12517.215,E2 -12517.215} C_VEL
LIN {X 0,Y 387.178,Z 423.128,A -85,B 0,C 180,E1 -12518.008,E2 -12518.008} C_VEL
LIN {X 0,Y 384.673,Z 421.95,A -85,B 0,C 180,E1 -12519.199,E2 -12519.199} C_VEL
LIN {X 0,Y 382.481,Z 419.775,A -85,B 0,C 180,E1 -12520.187,E2 -12520.187} C_VEL
LIN {X 0,Y 381.134,Z 417.196,A -85,B 0,C 180,E1 -12520.792,E2 -12520.792} C_VEL
LIN {X 0,Y 378.39,Z 415.583,A -85,B 0,C 180,E1 -12521.789,E2 -12521.789} C_VEL
LIN {X 0,Y 376.729,Z 413.367,A -85,B 0,C 180,E1 -12522.405,E2 -12522.405} C_VEL
LIN {X 0,Y 376.109,Z 411.137,A -85,B 0,C 180,E1 -12522.718,E2 -12522.718} C_VEL
LIN {X 0,Y 376.025,Z 411.146,A -85,B 0,C 180,E1 -12526.281,E2 -12526.281} C_VEL
LIN {X 0,Y 375.994,Z 411.149,A -85,B 0,C 180,E1 -12529.661,E2 -12529.661} C_VEL
LIN {X 0,Y 375.992,Z 411.146,A -85,B 0,C 180,E1 -12533.668,E2 -12533.668} C_VEL
LIN {X 0,Y 376.016,Z 411.149,A -85,B 0,C 180,E1 -12536.652,E2 -12536.652} C_VEL
LIN {X 0,Y 375.966,Z 411.151,A -85,B 0,C 180,E1 -12539.079,E2 -12539.079} C_VEL
LIN {X 0,Y 375.945,Z 411.155,A -85,B 0,C 180,E1 -12542.829,E2 -12542.829} C_VEL
LIN {X 0,Y 375.954,Z 411.151,A -85,B 0,C 180,E1 -12545.416,E2 -12545.416} C_VEL
LIN {X 0,Y 375.973,Z 411.154,A -85,B 0,C 180,E1 -12548.271,E2 -12548.271} C_VEL
LIN {X 0,Y 375.992,Z 411.148,A -85,B 0,C 180,E1 -12550.035,E2 -12550.035} C_VEL
LIN {X 0,Y 375.294,Z 411.236,A -85,B 0,C 180,E1 -12550.929,E2 -12550.929} C_VEL
LIN {X 0,Y 372.401,Z 411.6,A -85,B 0,C 180,E1 -12552.382,E2 -12552.382} C_VEL
LIN {X 0,Y 369.995,Z 411.894,A -85,B 0,C 180,E1 -12553.557,E2 -12553.557} C_VEL
LIN {X 0,Y 369.004,Z 412.021,A -85,B 0,C 180,E1 -12554.466,E2 -12554.466} C_VEL
LIN {X 0,Y 368.946,Z 412.025,A -85,B 0,C 180,E1 -12554.773,E2 -12554.773} C_VEL
LIN {X 0,Y 368.878,Z 412.038,A -85,B 0,C 180,E1 -12558.178,E2 -12558.178} C_VEL
LIN {X 0,Y 368.905,Z 412.029,A -85,B 0,C 180,E1 -12561.36,E2 -12561.36} C_VEL
LIN {X 0,Y 368.932,Z 412.026,A -85,B 0,C 180,E1 -12565.147,E2 -12565.147} C_VEL
LIN {X 0,Y 368.925,Z 412.027,A -85,B 0,C 180,E1 -12569.047,E2 -12569.047} C_VEL
LIN {X 0,Y 368.982,Z 412.021,A -85,B 0,C 180,E1 -12571.565,E2 -12571.565} C_VEL
LIN {X 0,Y 368.953,Z 412.023,A -85,B 0,C 180,E1 -12575.225,E2 -12575.225} C_VEL
LIN {X 0,Y 368.933,Z 412.025,A -85,B 0,C 180,E1 -12578.974,E2 -12578.974} C_VEL
LIN {X 0,Y 368.987,Z 412.021,A -85,B 0,C 180,E1 -12582.258,E2 -12582.258} C_VEL
LIN {X 0,Y 369.033,Z 412.015,A -85,B 0,C 180,E1 -12586.228,E2 -12586.228} C_VEL
LIN {X 0,Y 369.064,Z 412.012,A -85,B 0,C 180,E1 -12590.132,E2 -12590.132} C_VEL
LIN {X 0,Y 369.184,Z 411.995,A -85,B 0,C 180,E1 -12592.343,E2 -12592.343} C_VEL
LIN {X 0,Y 369.141,Z 412,A -85,B 0,C 180,E1 -12594.538,E2 -12594.538} C_VEL
LIN {X 0,Y 369.315,Z 411.982,A -85,B 0,C 180,E1 -12597.819,E2 -12597.819} C_VEL
LIN {X 0,Y 369.455,Z 411.963,A -85,B 0,C 180,E1 -12600.001,E2 -12600.001} C_VEL
LIN {X 0,Y 369.316,Z 411.979,A -85,B 0,C 180,E1 -12602.182,E2 -12602.182} C_VEL
LIN {X 0,Y 369.206,Z 411.991,A -85,B 0,C 180,E1 -12606.559,E2 -12606.559} C_VEL
LIN {X 0,Y 369.135,Z 412.001,A -85,B 0,C 180,E1 -12608.762,E2 -12608.762} C_VEL
LIN {X 0,Y 369.003,Z 412.017,A -85,B 0,C 180,E1 -12612.094,E2 -12612.094} C_VEL
LIN {X 0,Y 368.996,Z 412.023,A -85,B 0,C 180,E1 -12615.465,E2 -12615.465} C_VEL
LIN {X 0,Y 368.956,Z 412.025,A -85,B 0,C 180,E1 -12618.895,E2 -12618.895} C_VEL
LIN {X 0,Y 368.931,Z 412.026,A -85,B 0,C 180,E1 -12622.396,E2 -12622.396} C_VEL
LIN {X 0,Y 368.999,Z 412.018,A -85,B 0,C 180,E1 -12625.981,E2 -12625.981} C_VEL
LIN {X 0,Y 368.914,Z 412.029,A -85,B 0,C 180,E1 -12629.691,E2 -12629.691} C_VEL
LIN {X 0,Y 368.896,Z 412.036,A -85,B 0,C 180,E1 -12633.044,E2 -12633.044} C_VEL
LIN {X 0,Y 368.918,Z 412.032,A -85,B 0,C 180,E1 -12636.197,E2 -12636.197} C_VEL
LIN {X 0,Y 368.936,Z 412.198,A -85,B 0,C 180,E1 -12637.56,E2 -12637.56} C_VEL
LIN {X 0,Y 369.298,Z 414.539,A -85,B 0,C 180,E1 -12640.428,E2 -12640.428} C_VEL
LIN {X 0,Y 369.724,Z 417.522,A -85,B 0,C 180,E1 -12643.753,E2 -12643.753} C_VEL
LIN {X 0,Y 370.093,Z 420.578,A -85,B 0,C 180,E1 -12646.872,E2 -12646.872} C_VEL
LIN {X 0,Y 370.059,Z 423.691,A -85,B 0,C 180,E1 -12649.781,E2 -12649.781} C_VEL
LIN {X 0,Y 369.615,Z 427.396,A -85,B 0,C 180,E1 -12652.998,E2 -12652.998} C_VEL
LIN {X 0,Y 369.11,Z 431.671,A -85,B 0,C 180,E1 -12656.484,E2 -12656.484} C_VEL
LIN {X 0,Y 368.667,Z 436.578,A -85,B 0,C 180,E1 -12660.288,E2 -12660.288} C_VEL
LIN {X 0,Y 368.313,Z 441.579,A -85,B 0,C 180,E1 -12663.968,E2 -12663.968} C_VEL
LIN {X 0,Y 367.96,Z 446.597,A -85,B 0,C 180,E1 -12667.543,E2 -12667.543} C_VEL
LIN {X 0,Y 367.762,Z 450.609,A -85,B 0,C 180,E1 -12670.317,E2 -12670.317} C_VEL
LIN {X 0,Y 370.974,Z 466.374,A -85,B 0,C 180,E1 -12671.096,E2 -12671.096} C_VEL
LIN {X 0,Y 372.833,Z 478.671,A -85,B 0,C 180,E1 -12671.912,E2 -12671.912} C_VEL
LIN {X 0,Y 373.592,Z 486.122,A -85,B 0,C 180,E1 -12672.483,E2 -12672.483} C_VEL
LIN {X 0,Y 372.624,Z 497.035,A -85,B 0,C 180,E1 -12673.425,E2 -12673.425} C_VEL
LIN {X 0,Y 371.734,Z 505.982,A -85,B 0,C 180,E1 -12674.371,E2 -12674.371} C_VEL
LIN {X 0,Y 371.043,Z 513.734,A -85,B 0,C 180,E1 -12675.35,E2 -12675.35} C_VEL
LIN {X 0,Y 370.249,Z 521.742,A -85,B 0,C 180,E1 -12676.554,E2 -12676.554} C_VEL
LIN {X 0,Y 369.519,Z 527.944,A -85,B 0,C 180,E1 -12677.645,E2 -12677.645} C_VEL
LIN {X 0,Y 368.837,Z 534.484,A -85,B 0,C 180,E1 -12679.015,E2 -12679.015} C_VEL
LIN {X 0,Y 368.413,Z 538.989,A -85,B 0,C 180,E1 -12680.114,E2 -12680.114} C_VEL
LIN {X 0,Y 367.912,Z 544.483,A -85,B 0,C 180,E1 -12681.763,E2 -12681.763} C_VEL
LIN {X 0,Y 367.63,Z 548.81,A -85,B 0,C 180,E1 -12683.413,E2 -12683.413} C_VEL
LIN {X 0,Y 367.504,Z 551.178,A -85,B 0,C 180,E1 -12684.513,E2 -12684.513} C_VEL
LIN {X 0,Y 367.475,Z 552.979,A -85,B 0,C 180,E1 -12685.612,E2 -12685.612} C_VEL
LIN {X 0,Y 367.359,Z 555.424,A -85,B 0,C 180,E1 -12687.807,E2 -12687.807} C_VEL
LIN {X 0,Y 367.392,Z 556.014,A -85,B 0,C 180,E1 -12688.904,E2 -12688.904} C_VEL
LIN {X 0,Y 367.392,Z 556.015,A -85,B 0,C 180,E1 -12691.096,E2 -12691.096} C_VEL
LIN {X 0,Y 367.358,Z 555.425,A -85,B 0,C 180,E1 -12692.193,E2 -12692.193} C_VEL
LIN {X 0,Y 367.475,Z 552.98,A -85,B 0,C 180,E1 -12694.387,E2 -12694.387} C_VEL
LIN {X 0,Y 367.552,Z 549.85,A -85,B 0,C 180,E1 -12696.117,E2 -12696.117} C_VEL
LIN {X 0,Y 367.793,Z 546.039,A -85,B 0,C 180,E1 -12697.687,E2 -12697.687} C_VEL
LIN {X 0,Y 368.23,Z 540.907,A -85,B 0,C 180,E1 -12699.336,E2 -12699.336} C_VEL
LIN {X 0,Y 368.752,Z 535.644,A -85,B 0,C 180,E1 -12700.709,E2 -12700.709} C_VEL
LIN {X 0,Y 369.343,Z 529.322,A -85,B 0,C 180,E1 -12702.082,E2 -12702.082} C_VEL
LIN {X 0,Y 370.033,Z 523.371,A -85,B 0,C 180,E1 -12703.174,E2 -12703.174} C_VEL
LIN {X 0,Y 370.858,Z 515.133,A -85,B 0,C 180,E1 -12704.452,E2 -12704.452} C_VEL
LIN {X 0,Y 371.62,Z 507.121,A -85,B 0,C 180,E1 -12705.493,E2 -12705.493} C_VEL
LIN {X 0,Y 372.455,Z 498.391,A -85,B 0,C 180,E1 -12706.441,E2 -12706.441} C_VEL
LIN {X 0,Y 373.291,Z 489.394,A -85,B 0,C 180,E1 -12707.249,E2 -12707.249} C_VEL
LIN {X 0,Y 373.526,Z 483.759,A -85,B 0,C 180,E1 -12707.698,E2 -12707.698} C_VEL
LIN {X 0,Y 372.01,Z 472.806,A -85,B 0,C 180,E1 -12708.496,E2 -12708.496} C_VEL
LIN {X 0,Y 370.095,Z 461.947,A -85,B 0,C 180,E1 -12709.139,E2 -12709.139} C_VEL
LIN {X 0,Y 367.825,Z 451.383,A -85,B 0,C 180,E1 -12709.635,E2 -12709.635} C_VEL
LIN {X 0,Y 367.764,Z 450.614,A -85,B 0,C 180,E1 -12709.679,E2 -12709.679} C_VEL
LIN {X 0,Y 368.062,Z 444.909,A -85,B 0,C 180,E1 -12713.639,E2 -12713.639} C_VEL
LIN {X 0,Y 368.39,Z 439.894,A -85,B 0,C 180,E1 -12717.249,E2 -12717.249} C_VEL
LIN {X 0,Y 368.82,Z 434.932,A -85,B 0,C 180,E1 -12720.963,E2 -12720.963} C_VEL
LIN {X 0,Y 369.329,Z 430.05,A -85,B 0,C 180,E1 -12724.81,E2 -12724.81} C_VEL
LIN {X 0,Y 369.675,Z 426.838,A -85,B 0,C 180,E1 -12727.47,E2 -12727.47} C_VEL
LIN {X 0,Y 370.083,Z 423.28,A -85,B 0,C 180,E1 -12730.569,E2 -12730.569} C_VEL
LIN {X 0,Y 370.09,Z 420.556,A -85,B 0,C 180,E1 -12733.128,E2 -12733.128} C_VEL
LIN {X 0,Y 369.723,Z 417.511,A -85,B 0,C 180,E1 -12736.246,E2 -12736.246} C_VEL
LIN {X 0,Y 369.282,Z 414.45,A -85,B 0,C 180,E1 -12739.678,E2 -12739.678} C_VEL
LIN {X 0,Y 368.934,Z 412.195,A -85,B 0,C 180,E1 -12742.44,E2 -12742.44} C_VEL
LIN {X 0,Y 368.934,Z 412.031,A -85,B 0,C 180,E1 -12745.146,E2 -12745.146} C_VEL
LIN {X 0,Y 368.926,Z 412.031,A -85,B 0,C 180,E1 -12749.046,E2 -12749.046} C_VEL
LIN {X 0,Y 368.984,Z 412.02,A -85,B 0,C 180,E1 -12751.564,E2 -12751.564} C_VEL
LIN {X 0,Y 368.954,Z 412.025,A -85,B 0,C 180,E1 -12755.224,E2 -12755.224} C_VEL
LIN {X 0,Y 368.933,Z 412.029,A -85,B 0,C 180,E1 -12758.972,E2 -12758.972} C_VEL
LIN {X 0,Y 368.986,Z 412.021,A -85,B 0,C 180,E1 -12762.256,E2 -12762.256} C_VEL
LIN {X 0,Y 369.032,Z 412.016,A -85,B 0,C 180,E1 -12766.227,E2 -12766.227} C_VEL
LIN {X 0,Y 369.062,Z 412.012,A -85,B 0,C 180,E1 -12770.131,E2 -12770.131} C_VEL
LIN {X 0,Y 369.183,Z 411.999,A -85,B 0,C 180,E1 -12772.342,E2 -12772.342} C_VEL
LIN {X 0,Y 369.139,Z 412.006,A -85,B 0,C 180,E1 -12774.537,E2 -12774.537} C_VEL
LIN {X 0,Y 369.313,Z 411.979,A -85,B 0,C 180,E1 -12777.818,E2 -12777.818} C_VEL
LIN {X 0,Y 369.452,Z 411.963,A -85,B 0,C 180,E1 -12779.999,E2 -12779.999} C_VEL
LIN {X 0,Y 369.313,Z 411.983,A -85,B 0,C 180,E1 -12782.181,E2 -12782.181} C_VEL
LIN {X 0,Y 369.197,Z 411.996,A -85,B 0,C 180,E1 -12786.614,E2 -12786.614} C_VEL
LIN {X 0,Y 369.131,Z 412.002,A -85,B 0,C 180,E1 -12788.76,E2 -12788.76} C_VEL
LIN {X 0,Y 368.999,Z 412.023,A -85,B 0,C 180,E1 -12792.093,E2 -12792.093} C_VEL
LIN {X 0,Y 368.993,Z 412.019,A -85,B 0,C 180,E1 -12795.464,E2 -12795.464} C_VEL
LIN {X 0,Y 368.975,Z 412.02,A -85,B 0,C 180,E1 -12798.892,E2 -12798.892} C_VEL
LIN {X 0,Y 368.925,Z 412.029,A -85,B 0,C 180,E1 -12802.395,E2 -12802.395} C_VEL
LIN {X 0,Y 368.993,Z 412.025,A -85,B 0,C 180,E1 -12805.98,E2 -12805.98} C_VEL
LIN {X 0,Y 368.96,Z 412.022,A -85,B 0,C 180,E1 -12808.813,E2 -12808.813} C_VEL
LIN {X 0,Y 368.903,Z 412.032,A -85,B 0,C 180,E1 -12812.237,E2 -12812.237} C_VEL
LIN {X 0,Y 368.922,Z 412.027,A -85,B 0,C 180,E1 -12815.002,E2 -12815.002} C_VEL
LIN {X 0,Y 368.906,Z 412.029,A -85,B 0,C 180,E1 -12818.641,E2 -12818.641} C_VEL
LIN {X 0,Y 368.935,Z 412.029,A -85,B 0,C 180,E1 -12822.02,E2 -12822.02} C_VEL
LIN {X 0,Y 368.984,Z 412.021,A -85,B 0,C 180,E1 -12825.193,E2 -12825.193} C_VEL
LIN {X 0,Y 368.939,Z 412.026,A -85,B 0,C 180,E1 -12828.186,E2 -12828.186} C_VEL
LIN {X 0,Y 368.907,Z 412.033,A -85,B 0,C 180,E1 -12831.359,E2 -12831.359} C_VEL
LIN {X 0,Y 368.931,Z 412.028,A -85,B 0,C 180,E1 -12835.147,E2 -12835.147} C_VEL
LIN {X 0,Y 368.923,Z 412.029,A -85,B 0,C 180,E1 -12839.047,E2 -12839.047} C_VEL
LIN {X 0,Y 368.974,Z 412.025,A -85,B 0,C 180,E1 -12841.564,E2 -12841.564} C_VEL
LIN {X 0,Y 368.995,Z 412.019,A -85,B 0,C 180,E1 -12844.02,E2 -12844.02} C_VEL
LIN {X 0,Y 368.928,Z 412.03,A -85,B 0,C 180,E1 -12847.605,E2 -12847.605} C_VEL
LIN {X 0,Y 368.978,Z 412.025,A -85,B 0,C 180,E1 -12851.107,E2 -12851.107} C_VEL
LIN {X 0,Y 369.002,Z 412.023,A -85,B 0,C 180,E1 -12855.101,E2 -12855.101} C_VEL
LIN {X 0,Y 369.006,Z 412.027,A -85,B 0,C 180,E1 -12855.419,E2 -12855.419} C_VEL
LIN {X 0,Y 369.766,Z 414.395,A -85,B 0,C 180,E1 -12855.695,E2 -12855.695} C_VEL
LIN {X 0,Y 371.298,Z 416.379,A -85,B 0,C 180,E1 -12856.163,E2 -12856.163} C_VEL
LIN {X 0,Y 373.751,Z 418.119,A -85,B 0,C 180,E1 -12856.913,E2 -12856.913} C_VEL
LIN {X 0,Y 375.516,Z 420.998,A -85,B 0,C 180,E1 -12857.537,E2 -12857.537} C_VEL
LIN {X 0,Y 377.842,Z 423.109,A -85,B 0,C 180,E1 -12858.359,E2 -12858.359} C_VEL
LIN {X 0,Y 379.348,Z 424.072,A -85,B 0,C 180,E1 -12858.896,E2 -12858.896} C_VEL
LIN {X 0,Y 381.257,Z 426.948,A -85,B 0,C 180,E1 -12859.714,E2 -12859.714} C_VEL
LIN {X 0,Y 384.014,Z 429.238,A -85,B 0,C 180,E1 -12860.918,E2 -12860.918} C_VEL
LIN {X 0,Y 386.041,Z 430.344,A -85,B 0,C 180,E1 -12861.883,E2 -12861.883} C_VEL
LIN {X 0,Y 387.777,Z 432.961,A -85,B 0,C 180,E1 -12862.928,E2 -12862.928} C_VEL
LIN {X 0,Y 389.811,Z 435.008,A -85,B 0,C 180,E1 -12864.309,E2 -12864.309} C_VEL
LIN {X 0,Y 391.644,Z 436.139,A -85,B 0,C 180,E1 -12865.884,E2 -12865.884} C_VEL
LIN {X 0,Y 393.22,Z 436.524,A -85,B 0,C 180,E1 -12867.952,E2 -12867.952} C_VEL
LIN {X 0,Y 393.637,Z 436.552,A -85,B 0,C 180,E1 -12868.977,E2 -12868.977} C_VEL
LIN {X 0,Y 393.779,Z 436.58,A -85,B 0,C 180,E1 -12870,E2 -12870} C_VEL
LIN {X 0,Y 393.63,Z 436.552,A -85,B 0,C 180,E1 -12871.061,E2 -12871.061} C_VEL
LIN {X 0,Y 392.567,Z 436.348,A -85,B 0,C 180,E1 -12873.079,E2 -12873.079} C_VEL
LIN {X 0,Y 391.09,Z 435.881,A -85,B 0,C 180,E1 -12874.639,E2 -12874.639} C_VEL
LIN {X 0,Y 389.048,Z 434.378,A -85,B 0,C 180,E1 -12876.223,E2 -12876.223} C_VEL
LIN {X 0,Y 386.934,Z 431.838,A -85,B 0,C 180,E1 -12877.579,E2 -12877.579} C_VEL
LIN {X 0,Y 385.902,Z 430.05,A -85,B 0,C 180,E1 -12878.206,E2 -12878.206} C_VEL
LIN {X 0,Y 383.076,Z 428.609,A -85,B 0,C 180,E1 -12879.504,E2 -12879.504} C_VEL
LIN {X 0,Y 380.566,Z 426.104,A -85,B 0,C 180,E1 -12880.575,E2 -12880.575} C_VEL
LIN {X 0,Y 379.094,Z 423.759,A -85,B 0,C 180,E1 -12881.205,E2 -12881.205} C_VEL
LIN {X 0,Y 376.335,Z 421.954,A -85,B 0,C 180,E1 -12882.162,E2 -12882.162} C_VEL
LIN {X 0,Y 374.319,Z 419.239,A -85,B 0,C 180,E1 -12882.888,E2 -12882.888} C_VEL
LIN {X 0,Y 373.606,Z 417.793,A -85,B 0,C 180,E1 -12883.139,E2 -12883.139} C_VEL
LIN {X 0,Y 370.977,Z 416.079,A -85,B 0,C 180,E1 -12883.937,E2 -12883.937} C_VEL
LIN {X 0,Y 369.459,Z 413.757,A -85,B 0,C 180,E1 -12884.405,E2 -12884.405} C_VEL
LIN {X 0,Y 369.016,Z 412.022,A -85,B 0,C 180,E1 -12884.617,E2 -12884.617} C_VEL
LIN {X 0,Y 368.997,Z 412.022,A -85,B 0,C 180,E1 -12887.769,E2 -12887.769} C_VEL
LIN {X 0,Y 368.925,Z 412.028,A -85,B 0,C 180,E1 -12891.22,E2 -12891.22} C_VEL
LIN {X 0,Y 368.954,Z 412.028,A -85,B 0,C 180,E1 -12894.775,E2 -12894.775} C_VEL
LIN {X 0,Y 368.964,Z 412.022,A -85,B 0,C 180,E1 -12897.203,E2 -12897.203} C_VEL
LIN {X 0,Y 368.915,Z 412.028,A -85,B 0,C 180,E1 -12899.69,E2 -12899.69} C_VEL
LIN {X 0,Y 368.892,Z 412.032,A -85,B 0,C 180,E1 -12903.043,E2 -12903.043} C_VEL
LIN {X 0,Y 368.914,Z 412.032,A -85,B 0,C 180,E1 -12906.197,E2 -12906.197} C_VEL
LIN {X 0,Y 368.919,Z 412.03,A -85,B 0,C 180,E1 -12910.048,E2 -12910.048} C_VEL
LIN {X 0,Y 368.934,Z 412.025,A -85,B 0,C 180,E1 -12913.297,E2 -12913.297} C_VEL
LIN {X 0,Y 368.946,Z 412.025,A -85,B 0,C 180,E1 -12914.773,E2 -12914.773} C_VEL
LIN {X 0,Y 368.324,Z 412.107,A -85,B 0,C 180,E1 -12915.684,E2 -12915.684} C_VEL
LIN {X 0,Y 365.438,Z 412.465,A -85,B 0,C 180,E1 -12917.163,E2 -12917.163} C_VEL
LIN {X 0,Y 362.965,Z 412.774,A -85,B 0,C 180,E1 -12918.36,E2 -12918.36} C_VEL
LIN {X 0,Y 361.909,Z 412.901,A -85,B 0,C 180,E1 -12919.287,E2 -12919.287} C_VEL
LIN {X 0,Y 361.828,Z 412.911,A -85,B 0,C 180,E1 -12919.601,E2 -12919.601} C_VEL
LIN {X 0,Y 361.868,Z 412.906,A -85,B 0,C 180,E1 -12922.983,E2 -12922.983} C_VEL
LIN {X 0,Y 361.859,Z 412.908,A -85,B 0,C 180,E1 -12926.63,E2 -12926.63} C_VEL
LIN {X 0,Y 361.872,Z 412.907,A -85,B 0,C 180,E1 -12929.673,E2 -12929.673} C_VEL
LIN {X 0,Y 361.95,Z 412.897,A -85,B 0,C 180,E1 -12933.476,E2 -12933.476} C_VEL
LIN {X 0,Y 361.886,Z 412.904,A -85,B 0,C 180,E1 -12937.145,E2 -12937.145} C_VEL
LIN {X 0,Y 361.917,Z 412.9,A -85,B 0,C 180,E1 -12940.725,E2 -12940.725} C_VEL
LIN {X 0,Y 361.944,Z 412.899,A -85,B 0,C 180,E1 -12944.227,E2 -12944.227} C_VEL
LIN {X 0,Y 361.995,Z 412.89,A -85,B 0,C 180,E1 -12946.528,E2 -12946.528} C_VEL
LIN {X 0,Y 362.027,Z 412.89,A -85,B 0,C 180,E1 -12949.939,E2 -12949.939} C_VEL
LIN {X 0,Y 362.147,Z 412.873,A -85,B 0,C 180,E1 -12952.193,E2 -12952.193} C_VEL
LIN {X 0,Y 362.115,Z 412.875,A -85,B 0,C 180,E1 -12954.432,E2 -12954.432} C_VEL
LIN {X 0,Y 362.279,Z 412.859,A -85,B 0,C 180,E1 -12957.777,E2 -12957.777} C_VEL
LIN {X 0,Y 362.425,Z 412.839,A -85,B 0,C 180,E1 -12960.001,E2 -12960.001} C_VEL
LIN {X 0,Y 362.28,Z 412.855,A -85,B 0,C 180,E1 -12962.224,E2 -12962.224} C_VEL
LIN {X 0,Y 362.169,Z 412.868,A -85,B 0,C 180,E1 -12966.687,E2 -12966.687} C_VEL
LIN {X 0,Y 362.072,Z 412.882,A -85,B 0,C 180,E1 -12968.934,E2 -12968.934} C_VEL
LIN {X 0,Y 361.958,Z 412.894,A -85,B 0,C 180,E1 -12972.333,E2 -12972.333} C_VEL
LIN {X 0,Y 361.96,Z 412.894,A -85,B 0,C 180,E1 -12974.621,E2 -12974.621} C_VEL
LIN {X 0,Y 361.954,Z 412.895,A -85,B 0,C 180,E1 -12978.1,E2 -12978.1} C_VEL
LIN {X 0,Y 361.89,Z 412.905,A -85,B 0,C 180,E1 -12981.654,E2 -12981.654} C_VEL
LIN {X 0,Y 361.927,Z 412.904,A -85,B 0,C 180,E1 -12985.291,E2 -12985.291} C_VEL
LIN {X 0,Y 361.907,Z 412.902,A -85,B 0,C 180,E1 -12987.78,E2 -12987.78} C_VEL
LIN {X 0,Y 361.837,Z 412.911,A -85,B 0,C 180,E1 -12991.63,E2 -12991.63} C_VEL
LIN {X 0,Y 361.874,Z 412.911,A -85,B 0,C 180,E1 -12995.346,E2 -12995.346} C_VEL
LIN {X 0,Y 361.902,Z 413.117,A -85,B 0,C 180,E1 -12997.232,E2 -12997.232} C_VEL
LIN {X 0,Y 362.337,Z 416.038,A -85,B 0,C 180,E1 -13000.848,E2 -13000.848} C_VEL
LIN {X 0,Y 362.763,Z 419.036,A -85,B 0,C 180,E1 -13004.223,E2 -13004.223} C_VEL
LIN {X 0,Y 363.084,Z 422.096,A -85,B 0,C 180,E1 -13007.354,E2 -13007.354} C_VEL
LIN {X 0,Y 362.948,Z 425.203,A -85,B 0,C 180,E1 -13010.283,E2 -13010.283} C_VEL
LIN {X 0,Y 362.549,Z 428.366,A -85,B 0,C 180,E1 -13013.064,E2 -13013.064} C_VEL
LIN {X 0,Y 362.049,Z 432.602,A -85,B 0,C 180,E1 -13016.586,E2 -13016.586} C_VEL
LIN {X 0,Y 361.656,Z 436.464,A -85,B 0,C 180,E1 -13019.652,E2 -13019.652} C_VEL
LIN {X 0,Y 361.283,Z 441.519,A -85,B 0,C 180,E1 -13023.488,E2 -13023.488} C_VEL
LIN {X 0,Y 360.913,Z 446.436,A -85,B 0,C 180,E1 -13027.079,E2 -13027.079} C_VEL
LIN {X 0,Y 360.718,Z 450.54,A -85,B 0,C 180,E1 -13029.944,E2 -13029.944} C_VEL
LIN {X 0,Y 362.936,Z 460.982,A -85,B 0,C 180,E1 -13030.437,E2 -13030.437} C_VEL
LIN {X 0,Y 364.663,Z 470.45,A -85,B 0,C 180,E1 -13030.998,E2 -13030.998} C_VEL
LIN {X 0,Y 366.052,Z 480.192,A -85,B 0,C 180,E1 -13031.69,E2 -13031.69} C_VEL
LIN {X 0,Y 366.777,Z 485.909,A -85,B 0,C 180,E1 -13032.147,E2 -13032.147} C_VEL
LIN {X 0,Y 365.818,Z 496.824,A -85,B 0,C 180,E1 -13033.107,E2 -13033.107} C_VEL
LIN {X 0,Y 364.885,Z 505.77,A -85,B 0,C 180,E1 -13034.07,E2 -13034.07} C_VEL
LIN {X 0,Y 364.063,Z 514.324,A -85,B 0,C 180,E1 -13035.183,E2 -13035.183} C_VEL
LIN {X 0,Y 363.312,Z 521.529,A -85,B 0,C 180,E1 -13036.292,E2 -13036.292} C_VEL
LIN {X 0,Y 362.573,Z 527.732,A -85,B 0,C 180,E1 -13037.404,E2 -13037.404} C_VEL
LIN {X 0,Y 361.817,Z 534.271,A -85,B 0,C 180,E1 -13038.799,E2 -13038.799} C_VEL
LIN {X 0,Y 361.379,Z 538.776,A -85,B 0,C 180,E1 -13039.92,E2 -13039.92} C_VEL
LIN {X 0,Y 360.853,Z 544.27,A -85,B 0,C 180,E1 -13041.601,E2 -13041.601} C_VEL
LIN {X 0,Y 360.57,Z 548.599,A -85,B 0,C 180,E1 -13043.284,E2 -13043.284} C_VEL
LIN {X 0,Y 360.423,Z 550.967,A -85,B 0,C 180,E1 -13044.405,E2 -13044.405} C_VEL
LIN {X 0,Y 360.385,Z 552.768,A -85,B 0,C 180,E1 -13045.526,E2 -13045.526} C_VEL
LIN {X 0,Y 360.263,Z 555.213,A -85,B 0,C 180,E1 -13047.764,E2 -13047.764} C_VEL
LIN {X 0,Y 360.293,Z 555.803,A -85,B 0,C 180,E1 -13048.882,E2 -13048.882} C_VEL
LIN {X 0,Y 360.293,Z 555.803,A -85,B 0,C 180,E1 -13051.117,E2 -13051.117} C_VEL
LIN {X 0,Y 360.263,Z 555.213,A -85,B 0,C 180,E1 -13052.236,E2 -13052.236} C_VEL
LIN {X 0,Y 360.385,Z 552.768,A -85,B 0,C 180,E1 -13054.474,E2 -13054.474} C_VEL
LIN {X 0,Y 360.46,Z 549.975,A -85,B 0,C 180,E1 -13056.082,E2 -13056.082} C_VEL
LIN {X 0,Y 360.729,Z 545.826,A -85,B 0,C 180,E1 -13057.838,E2 -13057.838} C_VEL
LIN {X 0,Y 361.182,Z 540.695,A -85,B 0,C 180,E1 -13059.52,E2 -13059.52} C_VEL
LIN {X 0,Y 361.72,Z 535.43,A -85,B 0,C 180,E1 -13060.919,E2 -13060.919} C_VEL
LIN {X 0,Y 362.391,Z 529.111,A -85,B 0,C 180,E1 -13062.317,E2 -13062.317} C_VEL
LIN {X 0,Y 363.085,Z 523.159,A -85,B 0,C 180,E1 -13063.431,E2 -13063.431} C_VEL
LIN {X 0,Y 363.815,Z 516.228,A -85,B 0,C 180,E1 -13064.544,E2 -13064.544} C_VEL
LIN {X 0,Y 364.647,Z 508.045,A -85,B 0,C 180,E1 -13065.654,E2 -13065.654} C_VEL
LIN {X 0,Y 365.493,Z 499.531,A -85,B 0,C 180,E1 -13066.62,E2 -13066.62} C_VEL
LIN {X 0,Y 366.372,Z 490.815,A -85,B 0,C 180,E1 -13067.441,E2 -13067.441} C_VEL
LIN {X 0,Y 366.701,Z 484.88,A -85,B 0,C 180,E1 -13067.941,E2 -13067.941} C_VEL
LIN {X 0,Y 365,Z 472.586,A -85,B 0,C 180,E1 -13068.864,E2 -13068.864} C_VEL
LIN {X 0,Y 363.054,Z 461.688,A -85,B 0,C 180,E1 -13069.527,E2 -13069.527} C_VEL
LIN {X 0,Y 360.823,Z 451.41,A -85,B 0,C 180,E1 -13070.026,E2 -13070.026} C_VEL
LIN {X 0,Y 360.709,Z 450.389,A -85,B 0,C 180,E1 -13070.084,E2 -13070.084} C_VEL
LIN {X 0,Y 361.016,Z 444.747,A -85,B 0,C 180,E1 -13074.13,E2 -13074.13} C_VEL
LIN {X 0,Y 361.385,Z 439.76,A -85,B 0,C 180,E1 -13077.822,E2 -13077.822} C_VEL
LIN {X 0,Y 361.815,Z 434.824,A -85,B 0,C 180,E1 -13081.631,E2 -13081.631} C_VEL
LIN {X 0,Y 362.331,Z 430.138,A -85,B 0,C 180,E1 -13085.446,E2 -13085.446} C_VEL
LIN {X 0,Y 362.756,Z 426.775,A -85,B 0,C 180,E1 -13088.313,E2 -13088.313} C_VEL
LIN {X 0,Y 363.079,Z 423.624,A -85,B 0,C 180,E1 -13091.156,E2 -13091.156} C_VEL
LIN {X 0,Y 362.957,Z 420.495,A -85,B 0,C 180,E1 -13094.238,E2 -13094.238} C_VEL
LIN {X 0,Y 362.535,Z 417.513,A -85,B 0,C 180,E1 -13097.446,E2 -13097.446} C_VEL
LIN {X 0,Y 362.112,Z 414.562,A -85,B 0,C 180,E1 -13100.925,E2 -13100.925} C_VEL
LIN {X 0,Y 361.874,Z 412.96,A -85,B 0,C 180,E1 -13102.982,E2 -13102.982} C_VEL
LIN {X 0,Y 361.86,Z 412.911,A -85,B 0,C 180,E1 -13106.629,E2 -13106.629} C_VEL
LIN {X 0,Y 361.874,Z 412.905,A -85,B 0,C 180,E1 -13109.671,E2 -13109.671} C_VEL
LIN {X 0,Y 361.951,Z 412.896,A -85,B 0,C 180,E1 -13113.474,E2 -13113.474} C_VEL
LIN {X 0,Y 361.886,Z 412.906,A -85,B 0,C 180,E1 -13117.144,E2 -13117.144} C_VEL
LIN {X 0,Y 361.902,Z 412.908,A -85,B 0,C 180,E1 -13120.723,E2 -13120.723} C_VEL
LIN {X 0,Y 361.928,Z 412.9,A -85,B 0,C 180,E1 -13123.065,E2 -13123.065} C_VEL
LIN {X 0,Y 361.994,Z 412.896,A -85,B 0,C 180,E1 -13126.527,E2 -13126.527} C_VEL
LIN {X 0,Y 362.026,Z 412.887,A -85,B 0,C 180,E1 -13129.937,E2 -13129.937} C_VEL
LIN {X 0,Y 362.141,Z 412.875,A -85,B 0,C 180,E1 -13132.192,E2 -13132.192} C_VEL
LIN {X 0,Y 362.113,Z 412.881,A -85,B 0,C 180,E1 -13134.431,E2 -13134.431} C_VEL
LIN {X 0,Y 362.277,Z 412.855,A -85,B 0,C 180,E1 -13137.776,E2 -13137.776} C_VEL
LIN {X 0,Y 362.422,Z 412.839,A -85,B 0,C 180,E1 -13139.999,E2 -13139.999} C_VEL
LIN {X 0,Y 362.277,Z 412.86,A -85,B 0,C 180,E1 -13142.223,E2 -13142.223} C_VEL
LIN {X 0,Y 362.165,Z 412.871,A -85,B 0,C 180,E1 -13146.686,E2 -13146.686} C_VEL
LIN {X 0,Y 362.067,Z 412.881,A -85,B 0,C 180,E1 -13148.933,E2 -13148.933} C_VEL
LIN {X 0,Y 361.954,Z 412.9,A -85,B 0,C 180,E1 -13152.332,E2 -13152.332} C_VEL
LIN {X 0,Y 361.956,Z 412.897,A -85,B 0,C 180,E1 -13154.62,E2 -13154.62} C_VEL
LIN {X 0,Y 361.953,Z 412.901,A -85,B 0,C 180,E1 -13158.099,E2 -13158.099} C_VEL
LIN {X 0,Y 361.885,Z 412.906,A -85,B 0,C 180,E1 -13161.653,E2 -13161.653} C_VEL
LIN {X 0,Y 361.921,Z 412.9,A -85,B 0,C 180,E1 -13165.29,E2 -13165.29} C_VEL
LIN {X 0,Y 361.916,Z 412.904,A -85,B 0,C 180,E1 -13167.778,E2 -13167.778} C_VEL
LIN {X 0,Y 361.853,Z 412.911,A -85,B 0,C 180,E1 -13171.627,E2 -13171.627} C_VEL
LIN {X 0,Y 361.868,Z 412.907,A -85,B 0,C 180,E1 -13175.345,E2 -13175.345} C_VEL
LIN {X 0,Y 361.868,Z 412.906,A -85,B 0,C 180,E1 -13179.028,E2 -13179.028} C_VEL
LIN {X 0,Y 361.88,Z 412.905,A -85,B 0,C 180,E1 -13182.441,E2 -13182.441} C_VEL
LIN {X 0,Y 361.922,Z 412.903,A -85,B 0,C 180,E1 -13185.929,E2 -13185.929} C_VEL
LIN {X 0,Y 361.9,Z 412.904,A -85,B 0,C 180,E1 -13189.232,E2 -13189.232} C_VEL
LIN {X 0,Y 361.863,Z 412.907,A -85,B 0,C 180,E1 -13192.982,E2 -13192.982} C_VEL
LIN {X 0,Y 361.853,Z 412.908,A -85,B 0,C 180,E1 -13196.631,E2 -13196.631} C_VEL
LIN {X 0,Y 361.869,Z 412.91,A -85,B 0,C 180,E1 -13199.672,E2 -13199.672} C_VEL
LIN {X 0,Y 361.949,Z 412.901,A -85,B 0,C 180,E1 -13203.475,E2 -13203.475} C_VEL
LIN {X 0,Y 361.885,Z 412.908,A -85,B 0,C 180,E1 -13207.145,E2 -13207.145} C_VEL
LIN {X 0,Y 361.916,Z 412.903,A -85,B 0,C 180,E1 -13210.724,E2 -13210.724} C_VEL
LIN {X 0,Y 361.967,Z 413.082,A -85,B 0,C 180,E1 -13213.794,E2 -13213.794} C_VEL
LIN {X 0,Y 362.87,Z 415.661,A -85,B 0,C 180,E1 -13214.083,E2 -13214.083} C_VEL
LIN {X 0,Y 365.069,Z 417.94,A -85,B 0,C 180,E1 -13214.656,E2 -13214.656} C_VEL
LIN {X 0,Y 366.273,Z 418.742,A -85,B 0,C 180,E1 -13214.978,E2 -13214.978} C_VEL
LIN {X 0,Y 368.15,Z 421.846,A -85,B 0,C 180,E1 -13215.561,E2 -13215.561} C_VEL
LIN {X 0,Y 371.007,Z 424.138,A -85,B 0,C 180,E1 -13216.385,E2 -13216.385} C_VEL
LIN {X 0,Y 374.12,Z 428.154,A -85,B 0,C 180,E1 -13217.417,E2 -13217.417} C_VEL
LIN {X 0,Y 377.045,Z 430.333,A -85,B 0,C 180,E1 -13218.416,E2 -13218.416} C_VEL
LIN {X 0,Y 380.048,Z 434.016,A -85,B 0,C 180,E1 -13219.613,E2 -13219.613} C_VEL
LIN {X 0,Y 382.713,Z 436.125,A -85,B 0,C 180,E1 -13220.747,E2 -13220.747} C_VEL
LIN {X 0,Y 384.656,Z 437.168,A -85,B 0,C 180,E1 -13221.639,E2 -13221.639} C_VEL
LIN {X 0,Y 386.831,Z 440.15,A -85,B 0,C 180,E1 -13222.91,E2 -13222.91} C_VEL
LIN {X 0,Y 388.899,Z 442.063,A -85,B 0,C 180,E1 -13224.296,E2 -13224.296} C_VEL
LIN {X 0,Y 390.755,Z 443.182,A -85,B 0,C 180,E1 -13225.875,E2 -13225.875} C_VEL
LIN {X 0,Y 392.358,Z 443.566,A -85,B 0,C 180,E1 -13227.947,E2 -13227.947} C_VEL
LIN {X 0,Y 392.776,Z 443.598,A -85,B 0,C 180,E1 -13228.975,E2 -13228.975} C_VEL
LIN {X 0,Y 392.914,Z 443.626,A -85,B 0,C 180,E1 -13230,E2 -13230} C_VEL
LIN {X 0,Y 392.776,Z 443.601,A -85,B 0,C 180,E1 -13231.025,E2 -13231.025} C_VEL
LIN {X 0,Y 391.691,Z 443.393,A -85,B 0,C 180,E1 -13233.086,E2 -13233.086} C_VEL
LIN {X 0,Y 390.205,Z 442.906,A -85,B 0,C 180,E1 -13234.649,E2 -13234.649} C_VEL
LIN {X 0,Y 387.984,Z 441.368,A -85,B 0,C 180,E1 -13236.338,E2 -13236.338} C_VEL
LIN {X 0,Y 385.689,Z 438.755,A -85,B 0,C 180,E1 -13237.759,E2 -13237.759} C_VEL
LIN {X 0,Y 384.28,Z 436.821,A -85,B 0,C 180,E1 -13238.546,E2 -13238.546} C_VEL
LIN {X 0,Y 381.444,Z 435.253,A -85,B 0,C 180,E1 -13239.813,E2 -13239.813} C_VEL
LIN {X 0,Y 378.636,Z 432.432,A -85,B 0,C 180,E1 -13240.963,E2 -13240.963} C_VEL
LIN {X 0,Y 377.324,Z 430.435,A -85,B 0,C 180,E1 -13241.493,E2 -13241.493} C_VEL
LIN {X 0,Y 374.338,Z 428.376,A -85,B 0,C 180,E1 -13242.51,E2 -13242.51} C_VEL
LIN {X 0,Y 371.832,Z 425.225,A -85,B 0,C 180,E1 -13243.343,E2 -13243.343} C_VEL
LIN {X 0,Y 370.87,Z 424.02,A -85,B 0,C 180,E1 -13243.658,E2 -13243.658} C_VEL
LIN {X 0,Y 368.272,Z 421.992,A -85,B 0,C 180,E1 -13244.403,E2 -13244.403} C_VEL
LIN {X 0,Y 366.378,Z 418.974,A -85,B 0,C 180,E1 -13244.987,E2 -13244.987} C_VEL
LIN {X 0,Y 365.292,Z 418.056,A -85,B 0,C 180,E1 -13245.289,E2 -13245.289} C_VEL
LIN {X 0,Y 363.21,Z 416.143,A -85,B 0,C 180,E1 -13245.825,E2 -13245.825} C_VEL
LIN {X 0,Y 362.124,Z 413.842,A -85,B 0,C 180,E1 -13246.145,E2 -13246.145} C_VEL
LIN {X 0,Y 361.932,Z 412.902,A -85,B 0,C 180,E1 -13246.245,E2 -13246.245} C_VEL
LIN {X 0,Y 361.917,Z 412.905,A -85,B 0,C 180,E1 -13249.276,E2 -13249.276} C_VEL
LIN {X 0,Y 361.887,Z 412.907,A -85,B 0,C 180,E1 -13252.855,E2 -13252.855} C_VEL
LIN {X 0,Y 361.938,Z 412.902,A -85,B 0,C 180,E1 -13256.722,E2 -13256.722} C_VEL
LIN {X 0,Y 361.87,Z 412.909,A -85,B 0,C 180,E1 -13260.328,E2 -13260.328} C_VEL
LIN {X 0,Y 361.85,Z 412.912,A -85,B 0,C 180,E1 -13264.281,E2 -13264.281} C_VEL
LIN {X 0,Y 361.861,Z 412.907,A -85,B 0,C 180,E1 -13267.224,E2 -13267.224} C_VEL
LIN {X 0,Y 361.902,Z 412.904,A -85,B 0,C 180,E1 -13270.769,E2 -13270.769} C_VEL
LIN {X 0,Y 361.899,Z 412.908,A -85,B 0,C 180,E1 -13274.355,E2 -13274.355} C_VEL
LIN {X 0,Y 361.832,Z 412.911,A -85,B 0,C 180,E1 -13277.568,E2 -13277.568} C_VEL
LIN {X 0,Y 361.828,Z 412.911,A -85,B 0,C 180,E1 -13279.601,E2 -13279.601} C_VEL
LIN {X 0,Y 361.181,Z 412.998,A -85,B 0,C 180,E1 -13280.53,E2 -13280.53} C_VEL
LIN {X 0,Y 358.351,Z 413.355,A -85,B 0,C 180,E1 -13282.041,E2 -13282.041} C_VEL
LIN {X 0,Y 355.94,Z 413.654,A -85,B 0,C 180,E1 -13283.263,E2 -13283.263} C_VEL
LIN {X 0,Y 354.897,Z 413.78,A -85,B 0,C 180,E1 -13284.209,E2 -13284.209} C_VEL
LIN {X 0,Y 354.809,Z 413.788,A -85,B 0,C 180,E1 -13284.529,E2 -13284.529} C_VEL
LIN {X 0,Y 354.794,Z 413.789,A -85,B 0,C 180,E1 -13287.668,E2 -13287.668} C_VEL
LIN {X 0,Y 354.865,Z 413.779,A -85,B 0,C 180,E1 -13290.622,E2 -13290.622} C_VEL
LIN {X 0,Y 354.895,Z 413.779,A -85,B 0,C 180,E1 -13294.173,E2 -13294.173} C_VEL
LIN {X 0,Y 354.83,Z 413.788,A -85,B 0,C 180,E1 -13297.894,E2 -13297.894} C_VEL
LIN {X 0,Y 354.919,Z 413.778,A -85,B 0,C 180,E1 -13301.892,E2 -13301.892} C_VEL
LIN {X 0,Y 354.939,Z 413.773,A -85,B 0,C 180,E1 -13305.982,E2 -13305.982} C_VEL
LIN {X 0,Y 354.974,Z 413.77,A -85,B 0,C 180,E1 -13309.736,E2 -13309.736} C_VEL
LIN {X 0,Y 355.11,Z 413.751,A -85,B 0,C 180,E1 -13312.037,E2 -13312.037} C_VEL
LIN {X 0,Y 355.089,Z 413.751,A -85,B 0,C 180,E1 -13314.321,E2 -13314.321} C_VEL
LIN {X 0,Y 355.243,Z 413.736,A -85,B 0,C 180,E1 -13317.733,E2 -13317.733} C_VEL
LIN {X 0,Y 355.394,Z 413.714,A -85,B 0,C 180,E1 -13320.001,E2 -13320.001} C_VEL
LIN {X 0,Y 355.243,Z 413.732,A -85,B 0,C 180,E1 -13322.268,E2 -13322.268} C_VEL
LIN {X 0,Y 355.135,Z 413.745,A -85,B 0,C 180,E1 -13326.82,E2 -13326.82} C_VEL
LIN {X 0,Y 355.013,Z 413.762,A -85,B 0,C 180,E1 -13329.113,E2 -13329.113} C_VEL
LIN {X 0,Y 354.919,Z 413.771,A -85,B 0,C 180,E1 -13332.582,E2 -13332.582} C_VEL
LIN {X 0,Y 354.887,Z 413.776,A -85,B 0,C 180,E1 -13336.097,E2 -13336.097} C_VEL
LIN {X 0,Y 354.9,Z 413.774,A -85,B 0,C 180,E1 -13338.473,E2 -13338.473} C_VEL
LIN {X 0,Y 354.833,Z 413.782,A -85,B 0,C 180,E1 -13342.107,E2 -13342.107} C_VEL
LIN {X 0,Y 354.898,Z 413.775,A -85,B 0,C 180,E1 -13345.828,E2 -13345.828} C_VEL
LIN {X 0,Y 354.817,Z 413.786,A -85,B 0,C 180,E1 -13349.683,E2 -13349.683} C_VEL
LIN {X 0,Y 354.806,Z 413.788,A -85,B 0,C 180,E1 -13353.703,E2 -13353.703} C_VEL
LIN {X 0,Y 354.8,Z 413.792,A -85,B 0,C 180,E1 -13356.46,E2 -13356.46} C_VEL
LIN {X 0,Y 355.155,Z 416.043,A -85,B 0,C 180,E1 -13359.489,E2 -13359.489} C_VEL
LIN {X 0,Y 355.586,Z 419.007,A -85,B 0,C 180,E1 -13363.006,E2 -13363.006} C_VEL
LIN {X 0,Y 355.96,Z 422.047,A -85,B 0,C 180,E1 -13366.289,E2 -13366.289} C_VEL
LIN {X 0,Y 356.006,Z 425.156,A -85,B 0,C 180,E1 -13369.349,E2 -13369.349} C_VEL
LIN {X 0,Y 355.626,Z 428.312,A -85,B 0,C 180,E1 -13372.232,E2 -13372.232} C_VEL
LIN {X 0,Y 355.216,Z 431.483,A -85,B 0,C 180,E1 -13374.987,E2 -13374.987} C_VEL
LIN {X 0,Y 354.685,Z 436.345,A -85,B 0,C 180,E1 -13378.99,E2 -13378.99} C_VEL
LIN {X 0,Y 354.254,Z 441.266,A -85,B 0,C 180,E1 -13382.852,E2 -13382.852} C_VEL
LIN {X 0,Y 353.885,Z 446.267,A -85,B 0,C 180,E1 -13386.597,E2 -13386.597} C_VEL
LIN {X 0,Y 353.667,Z 450.195,A -85,B 0,C 180,E1 -13389.517,E2 -13389.517} C_VEL
LIN {X 0,Y 356.041,Z 461.368,A -85,B 0,C 180,E1 -13390.068,E2 -13390.068} C_VEL
LIN {X 0,Y 357.917,Z 471.758,A -85,B 0,C 180,E1 -13390.713,E2 -13390.713} C_VEL
LIN {X 0,Y 359.413,Z 482.627,A -85,B 0,C 180,E1 -13391.532,E2 -13391.532} C_VEL
LIN {X 0,Y 359.875,Z 487.332,A -85,B 0,C 180,E1 -13391.939,E2 -13391.939} C_VEL
LIN {X 0,Y 358.988,Z 496.611,A -85,B 0,C 180,E1 -13392.776,E2 -13392.776} C_VEL
LIN {X 0,Y 358.047,Z 505.559,A -85,B 0,C 180,E1 -13393.757,E2 -13393.757} C_VEL
LIN {X 0,Y 357.282,Z 512.993,A -85,B 0,C 180,E1 -13394.725,E2 -13394.725} C_VEL
LIN {X 0,Y 356.385,Z 521.317,A -85,B 0,C 180,E1 -13396.021,E2 -13396.021} C_VEL
LIN {X 0,Y 355.619,Z 527.52,A -85,B 0,C 180,E1 -13397.154,E2 -13397.154} C_VEL
LIN {X 0,Y 354.808,Z 534.059,A -85,B 0,C 180,E1 -13398.575,E2 -13398.575} C_VEL
LIN {X 0,Y 354.357,Z 538.564,A -85,B 0,C 180,E1 -13399.718,E2 -13399.718} C_VEL
LIN {X 0,Y 353.816,Z 544.059,A -85,B 0,C 180,E1 -13401.432,E2 -13401.432} C_VEL
LIN {X 0,Y 353.506,Z 548.387,A -85,B 0,C 180,E1 -13403.149,E2 -13403.149} C_VEL
LIN {X 0,Y 353.332,Z 550.754,A -85,B 0,C 180,E1 -13404.292,E2 -13404.292} C_VEL
LIN {X 0,Y 353.299,Z 552.556,A -85,B 0,C 180,E1 -13405.436,E2 -13405.436} C_VEL
LIN {X 0,Y 353.172,Z 555.002,A -85,B 0,C 180,E1 -13407.719,E2 -13407.719} C_VEL
LIN {X 0,Y 353.194,Z 555.592,A -85,B 0,C 180,E1 -13408.86,E2 -13408.86} C_VEL
LIN {X 0,Y 353.194,Z 555.592,A -85,B 0,C 180,E1 -13411.14,E2 -13411.14} C_VEL
LIN {X 0,Y 353.172,Z 555.002,A -85,B 0,C 180,E1 -13412.281,E2 -13412.281} C_VEL
LIN {X 0,Y 353.299,Z 552.557,A -85,B 0,C 180,E1 -13414.564,E2 -13414.564} C_VEL
LIN {X 0,Y 353.371,Z 550.092,A -85,B 0,C 180,E1 -13416.05,E2 -13416.05} C_VEL
LIN {X 0,Y 353.549,Z 547.145,A -85,B 0,C 180,E1 -13417.424,E2 -13417.424} C_VEL
LIN {X 0,Y 353.979,Z 542.399,A -85,B 0,C 180,E1 -13419.139,E2 -13419.139} C_VEL
LIN {X 0,Y 354.615,Z 536.375,A -85,B 0,C 180,E1 -13420.852,E2 -13420.852} C_VEL
LIN {X 0,Y 355.251,Z 530.274,A -85,B 0,C 180,E1 -13422.278,E2 -13422.278} C_VEL
LIN {X 0,Y 355.967,Z 524.574,A -85,B 0,C 180,E1 -13423.413,E2 -13423.413} C_VEL
LIN {X 0,Y 356.932,Z 516.016,A -85,B 0,C 180,E1 -13424.831,E2 -13424.831} C_VEL
LIN {X 0,Y 357.796,Z 507.833,A -85,B 0,C 180,E1 -13425.961,E2 -13425.961} C_VEL
LIN {X 0,Y 358.681,Z 499.319,A -85,B 0,C 180,E1 -13426.945,E2 -13426.945} C_VEL
LIN {X 0,Y 359.583,Z 490.603,A -85,B 0,C 180,E1 -13427.781,E2 -13427.781} C_VEL
LIN {X 0,Y 359.85,Z 485.698,A -85,B 0,C 180,E1 -13428.209,E2 -13428.209} C_VEL
LIN {X 0,Y 358.242,Z 473.854,A -85,B 0,C 180,E1 -13429.148,E2 -13429.148} C_VEL
LIN {X 0,Y 356.166,Z 462.061,A -85,B 0,C 180,E1 -13429.895,E2 -13429.895} C_VEL
LIN {X 0,Y 353.839,Z 451.672,A -85,B 0,C 180,E1 -13430.425,E2 -13430.425} C_VEL
LIN {X 0,Y 353.659,Z 450.169,A -85,B 0,C 180,E1 -13430.502,E2 -13430.502} C_VEL
LIN {X 0,Y 353.945,Z 445.427,A -85,B 0,C 180,E1 -13434.022,E2 -13434.022} C_VEL
LIN {X 0,Y 354.246,Z 441.266,A -85,B 0,C 180,E1 -13437.148,E2 -13437.148} C_VEL
LIN {X 0,Y 354.682,Z 436.346,A -85,B 0,C 180,E1 -13441.009,E2 -13441.009} C_VEL
LIN {X 0,Y 355.214,Z 431.483,A -85,B 0,C 180,E1 -13445.013,E2 -13445.013} C_VEL
LIN {X 0,Y 355.625,Z 428.287,A -85,B 0,C 180,E1 -13447.779,E2 -13447.779} C_VEL
LIN {X 0,Y 356.001,Z 425.136,A -85,B 0,C 180,E1 -13450.651,E2 -13450.651} C_VEL
LIN {X 0,Y 355.959,Z 422.043,A -85,B 0,C 180,E1 -13453.711,E2 -13453.711} C_VEL
LIN {X 0,Y 355.578,Z 419.005,A -85,B 0,C 180,E1 -13456.995,E2 -13456.995} C_VEL
LIN {X 0,Y 355.157,Z 416.041,A -85,B 0,C 180,E1 -13460.51,E2 -13460.51} C_VEL
LIN {X 0,Y 354.798,Z 413.793,A -85,B 0,C 180,E1 -13463.54,E2 -13463.54} C_VEL
LIN {X 0,Y 354.828,Z 413.787,A -85,B 0,C 180,E1 -13466.317,E2 -13466.317} C_VEL
LIN {X 0,Y 354.851,Z 413.781,A -85,B 0,C 180,E1 -13470.321,E2 -13470.321} C_VEL
LIN {X 0,Y 354.896,Z 413.775,A -85,B 0,C 180,E1 -13474.172,E2 -13474.172} C_VEL
LIN {X 0,Y 354.83,Z 413.783,A -85,B 0,C 180,E1 -13477.893,E2 -13477.893} C_VEL
LIN {X 0,Y 354.918,Z 413.772,A -85,B 0,C 180,E1 -13481.891,E2 -13481.891} C_VEL
LIN {X 0,Y 354.938,Z 413.77,A -85,B 0,C 180,E1 -13485.98,E2 -13485.98} C_VEL
LIN {X 0,Y 354.973,Z 413.765,A -85,B 0,C 180,E1 -13489.735,E2 -13489.735} C_VEL
LIN {X 0,Y 355.123,Z 413.748,A -85,B 0,C 180,E1 -13492.036,E2 -13492.036} C_VEL
LIN {X 0,Y 355.087,Z 413.755,A -85,B 0,C 180,E1 -13494.32,E2 -13494.32} C_VEL
LIN {X 0,Y 355.24,Z 413.732,A -85,B 0,C 180,E1 -13497.732,E2 -13497.732} C_VEL
LIN {X 0,Y 355.391,Z 413.715,A -85,B 0,C 180,E1 -13499.999,E2 -13499.999} C_VEL
LIN {X 0,Y 355.24,Z 413.736,A -85,B 0,C 180,E1 -13502.267,E2 -13502.267} C_VEL
LIN {X 0,Y 355.132,Z 413.746,A -85,B 0,C 180,E1 -13506.819,E2 -13506.819} C_VEL
LIN {X 0,Y 355.009,Z 413.76,A -85,B 0,C 180,E1 -13509.112,E2 -13509.112} C_VEL
LIN {X 0,Y 354.914,Z 413.774,A -85,B 0,C 180,E1 -13512.58,E2 -13512.58} C_VEL
LIN {X 0,Y 354.885,Z 413.781,A -85,B 0,C 180,E1 -13516.095,E2 -13516.095} C_VEL
LIN {X 0,Y 354.9,Z 413.776,A -85,B 0,C 180,E1 -13518.471,E2 -13518.471} C_VEL
LIN {X 0,Y 354.828,Z 413.788,A -85,B 0,C 180,E1 -13522.106,E2 -13522.106} C_VEL
LIN {X 0,Y 354.892,Z 413.779,A -85,B 0,C 180,E1 -13525.827,E2 -13525.827} C_VEL
LIN {X 0,Y 354.848,Z 413.784,A -85,B 0,C 180,E1 -13529.678,E2 -13529.678} C_VEL
LIN {X 0,Y 354.824,Z 413.787,A -85,B 0,C 180,E1 -13533.682,E2 -13533.682} C_VEL
LIN {X 0,Y 354.795,Z 413.788,A -85,B 0,C 180,E1 -13536.459,E2 -13536.459} C_VEL
LIN {X 0,Y 354.817,Z 413.787,A -85,B 0,C 180,E1 -13539.424,E2 -13539.424} C_VEL
LIN {X 0,Y 354.836,Z 413.782,A -85,B 0,C 180,E1 -13542.877,E2 -13542.877} C_VEL
LIN {X 0,Y 354.86,Z 413.781,A -85,B 0,C 180,E1 -13546.119,E2 -13546.119} C_VEL
LIN {X 0,Y 354.851,Z 413.782,A -85,B 0,C 180,E1 -13549.189,E2 -13549.189} C_VEL
LIN {X 0,Y 354.803,Z 413.786,A -85,B 0,C 180,E1 -13552.402,E2 -13552.402} C_VEL
LIN {X 0,Y 354.806,Z 413.786,A -85,B 0,C 180,E1 -13554.941,E2 -13554.941} C_VEL
LIN {X 0,Y 354.787,Z 413.788,A -85,B 0,C 180,E1 -13558.405,E2 -13558.405} C_VEL
LIN {X 0,Y 354.845,Z 413.785,A -85,B 0,C 180,E1 -13561.619,E2 -13561.619} C_VEL
LIN {X 0,Y 354.894,Z 413.775,A -85,B 0,C 180,E1 -13564.173,E2 -13564.173} C_VEL
LIN {X 0,Y 354.83,Z 413.784,A -85,B 0,C 180,E1 -13567.894,E2 -13567.894} C_VEL
LIN {X 0,Y 354.918,Z 413.775,A -85,B 0,C 180,E1 -13571.892,E2 -13571.892} C_VEL
LIN {X 0,Y 354.912,Z 413.789,A -85,B 0,C 180,E1 -13572.333,E2 -13572.333} C_VEL
LIN {X 0,Y 355.752,Z 416.376,A -85,B 0,C 180,E1 -13572.588,E2 -13572.588} C_VEL
LIN {X 0,Y 357.644,Z 418.565,A -85,B 0,C 180,E1 -13573.045,E2 -13573.045} C_VEL
LIN {X 0,Y 358.962,Z 419.669,A -85,B 0,C 180,E1 -13573.351,E2 -13573.351} C_VEL
LIN {X 0,Y 360.937,Z 422.738,A -85,B 0,C 180,E1 -13573.886,E2 -13573.886} C_VEL
LIN {X 0,Y 363.793,Z 425.258,A -85,B 0,C 180,E1 -13574.617,E2 -13574.617} C_VEL
LIN {X 0,Y 366.162,Z 428.522,A -85,B 0,C 180,E1 -13575.303,E2 -13575.303} C_VEL
LIN {X 0,Y 369.419,Z 431.276,A -85,B 0,C 180,E1 -13576.223,E2 -13576.223} C_VEL
LIN {X 0,Y 372.187,Z 434.702,A -85,B 0,C 180,E1 -13577.118,E2 -13577.118} C_VEL
LIN {X 0,Y 375.824,Z 437.612,A -85,B 0,C 180,E1 -13578.343,E2 -13578.343} C_VEL
LIN {X 0,Y 378.294,Z 440.571,A -85,B 0,C 180,E1 -13579.294,E2 -13579.294} C_VEL
LIN {X 0,Y 381.408,Z 443.019,A -85,B 0,C 180,E1 -13580.585,E2 -13580.585} C_VEL
LIN {X 0,Y 383.283,Z 444.109,A -85,B 0,C 180,E1 -13581.432,E2 -13581.432} C_VEL
LIN {X 0,Y 385.714,Z 447.122,A -85,B 0,C 180,E1 -13582.781,E2 -13582.781} C_VEL
LIN {X 0,Y 387.686,Z 448.941,A -85,B 0,C 180,E1 -13584.078,E2 -13584.078} C_VEL
LIN {X 0,Y 389.596,Z 450.124,A -85,B 0,C 180,E1 -13585.603,E2 -13585.603} C_VEL
LIN {X 0,Y 390.814,Z 450.444,A -85,B 0,C 180,E1 -13586.908,E2 -13586.908} C_VEL
LIN {X 0,Y 391.493,Z 450.612,A -85,B 0,C 180,E1 -13587.943,E2 -13587.943} C_VEL
LIN {X 0,Y 391.912,Z 450.645,A -85,B 0,C 180,E1 -13588.973,E2 -13588.973} C_VEL
LIN {X 0,Y 392.049,Z 450.673,A -85,B 0,C 180,E1 -13590,E2 -13590} C_VEL
LIN {X 0,Y 391.912,Z 450.647,A -85,B 0,C 180,E1 -13591.028,E2 -13591.028} C_VEL
LIN {X 0,Y 391.493,Z 450.602,A -85,B 0,C 180,E1 -13592.058,E2 -13592.058} C_VEL
LIN {X 0,Y 389.865,Z 450.221,A -85,B 0,C 180,E1 -13594.135,E2 -13594.135} C_VEL
LIN {X 0,Y 387.986,Z 449.121,A -85,B 0,C 180,E1 -13595.718,E2 -13595.718} C_VEL
LIN {X 0,Y 385.835,Z 447.279,A -85,B 0,C 180,E1 -13597.14,E2 -13597.14} C_VEL
LIN {X 0,Y 383.281,Z 444.111,A -85,B 0,C 180,E1 -13598.568,E2 -13598.568} C_VEL
LIN {X 0,Y 379.537,Z 441.714,A -85,B 0,C 180,E1 -13600.199,E2 -13600.199} C_VEL
LIN {X 0,Y 376.615,Z 438.708,A -85,B 0,C 180,E1 -13601.363,E2 -13601.363} C_VEL
LIN {X 0,Y 375.165,Z 436.961,A -85,B 0,C 180,E1 -13601.892,E2 -13601.892} C_VEL
LIN {X 0,Y 372.031,Z 434.55,A -85,B 0,C 180,E1 -13602.93,E2 -13602.93} C_VEL
LIN {X 0,Y 369.237,Z 431.024,A -85,B 0,C 180,E1 -13603.833,E2 -13603.833} C_VEL
LIN {X 0,Y 365.514,Z 427.786,A -85,B 0,C 180,E1 -13604.886,E2 -13604.886} C_VEL
LIN {X 0,Y 363.341,Z 424.761,A -85,B 0,C 180,E1 -13605.501,E2 -13605.501} C_VEL
LIN {X 0,Y 360.539,Z 422.25,A -85,B 0,C 180,E1 -13606.221,E2 -13606.221} C_VEL
LIN {X 0,Y 358.64,Z 419.197,A -85,B 0,C 180,E1 -13606.73,E2 -13606.73} C_VEL
LIN {X 0,Y 356.271,Z 417.19,A -85,B 0,C 180,E1 -13607.28,E2 -13607.28} C_VEL
LIN {X 0,Y 355.062,Z 414.661,A -85,B 0,C 180,E1 -13607.608,E2 -13607.608} C_VEL
LIN {X 0,Y 354.921,Z 413.775,A -85,B 0,C 180,E1 -13607.693,E2 -13607.693} C_VEL
LIN {X 0,Y 354.837,Z 413.782,A -85,B 0,C 180,E1 -13611.427,E2 -13611.427} C_VEL
LIN {X 0,Y 354.858,Z 413.785,A -85,B 0,C 180,E1 -13614.576,E2 -13614.576} C_VEL
LIN {X 0,Y 354.88,Z 413.778,A -85,B 0,C 180,E1 -13617.096,E2 -13617.096} C_VEL
LIN {X 0,Y 354.85,Z 413.78,A -85,B 0,C 180,E1 -13619.679,E2 -13619.679} C_VEL
LIN {X 0,Y 354.802,Z 413.786,A -85,B 0,C 180,E1 -13623.702,E2 -13623.702} C_VEL
LIN {X 0,Y 354.796,Z 413.793,A -85,B 0,C 180,E1 -13626.459,E2 -13626.459} C_VEL
LIN {X 0,Y 354.82,Z 413.784,A -85,B 0,C 180,E1 -13629.424,E2 -13629.424} C_VEL
LIN {X 0,Y 354.832,Z 413.784,A -85,B 0,C 180,E1 -13632.876,E2 -13632.876} C_VEL
LIN {X 0,Y 354.779,Z 413.793,A -85,B 0,C 180,E1 -13636.107,E2 -13636.107} C_VEL
LIN {X 0,Y 354.772,Z 413.788,A -85,B 0,C 180,E1 -13639.6,E2 -13639.6} C_VEL
LIN {X 0,Y 354.808,Z 413.789,A -85,B 0,C 180,E1 -13642.402,E2 -13642.402} C_VEL
LIN {X 0,Y 354.809,Z 413.788,A -85,B 0,C 180,E1 -13644.529,E2 -13644.529} C_VEL
LIN {X 0,Y 354.122,Z 413.873,A -85,B 0,C 180,E1 -13645.476,E2 -13645.476} C_VEL
LIN {X 0,Y 351.234,Z 414.23,A -85,B 0,C 180,E1 -13647.016,E2 -13647.016} C_VEL
LIN {X 0,Y 348.821,Z 414.535,A -85,B 0,C 180,E1 -13648.263,E2 -13648.263} C_VEL
LIN {X 0,Y 347.821,Z 414.656,A -85,B 0,C 180,E1 -13649.227,E2 -13649.227} C_VEL
LIN {X 0,Y 347.759,Z 414.665,A -85,B 0,C 180,E1 -13649.554,E2 -13649.554} C_VEL
LIN {X 0,Y 347.848,Z 414.653,A -85,B 0,C 180,E1 -13652.745,E2 -13652.745} C_VEL
LIN {X 0,Y 347.784,Z 414.664,A -85,B 0,C 180,E1 -13656.162,E2 -13656.162} C_VEL
LIN {X 0,Y 347.813,Z 414.662,A -85,B 0,C 180,E1 -13659.91,E2 -13659.91} C_VEL
LIN {X 0,Y 347.863,Z 414.652,A -85,B 0,C 180,E1 -13662.36,E2 -13662.36} C_VEL
LIN {X 0,Y 347.894,Z 414.651,A -85,B 0,C 180,E1 -13665.971,E2 -13665.971} C_VEL
LIN {X 0,Y 347.925,Z 414.646,A -85,B 0,C 180,E1 -13669.526,E2 -13669.526} C_VEL
LIN {X 0,Y 348.071,Z 414.629,A -85,B 0,C 180,E1 -13671.875,E2 -13671.875} C_VEL
LIN {X 0,Y 348.064,Z 414.627,A -85,B 0,C 180,E1 -13674.206,E2 -13674.206} C_VEL
LIN {X 0,Y 348.205,Z 414.612,A -85,B 0,C 180,E1 -13677.687,E2 -13677.687} C_VEL
LIN {X 0,Y 348.343,Z 414.592,A -85,B 0,C 180,E1 -13680.001,E2 -13680.001} C_VEL
LIN {X 0,Y 348.205,Z 414.608,A -85,B 0,C 180,E1 -13682.314,E2 -13682.314} C_VEL
LIN {X 0,Y 348.105,Z 414.621,A -85,B 0,C 180,E1 -13686.958,E2 -13686.958} C_VEL
LIN {X 0,Y 347.926,Z 414.642,A -85,B 0,C 180,E1 -13690.475,E2 -13690.475} C_VEL
LIN {X 0,Y 347.897,Z 414.647,A -85,B 0,C 180,E1 -13694.151,E2 -13694.151} C_VEL
LIN {X 0,Y 347.889,Z 414.647,A -85,B 0,C 180,E1 -13698.291,E2 -13698.291} C_VEL
LIN {X 0,Y 347.787,Z 414.662,A -85,B 0,C 180,E1 -13701.636,E2 -13701.636} C_VEL
LIN {X 0,Y 347.812,Z 414.662,A -85,B 0,C 180,E1 -13705.109,E2 -13705.109} C_VEL
LIN {X 0,Y 347.807,Z 414.659,A -85,B 0,C 180,E1 -13707.695,E2 -13707.695} C_VEL
LIN {X 0,Y 347.749,Z 414.665,A -85,B 0,C 180,E1 -13710.349,E2 -13710.349} C_VEL
LIN {X 0,Y 347.748,Z 414.668,A -85,B 0,C 180,E1 -13714.044,E2 -13714.044} C_VEL
LIN {X 0,Y 347.771,Z 414.666,A -85,B 0,C 180,E1 -13716.066,E2 -13716.066} C_VEL
LIN {X 0,Y 348.213,Z 417.523,A -85,B 0,C 180,E1 -13719.919,E2 -13719.919} C_VEL
LIN {X 0,Y 348.642,Z 420.493,A -85,B 0,C 180,E1 -13723.474,E2 -13723.474} C_VEL
LIN {X 0,Y 348.957,Z 423.544,A -85,B 0,C 180,E1 -13726.784,E2 -13726.784} C_VEL
LIN {X 0,Y 348.905,Z 426.73,A -85,B 0,C 180,E1 -13729.946,E2 -13729.946} C_VEL
LIN {X 0,Y 348.349,Z 430.966,A -85,B 0,C 180,E1 -13733.805,E2 -13733.805} C_VEL
LIN {X 0,Y 347.866,Z 434.606,A -85,B 0,C 180,E1 -13736.942,E2 -13736.942} C_VEL
LIN {X 0,Y 347.434,Z 438.843,A -85,B 0,C 180,E1 -13740.439,E2 -13740.439} C_VEL
LIN {X 0,Y 347.109,Z 442.777,A -85,B 0,C 180,E1 -13743.549,E2 -13743.549} C_VEL
LIN {X 0,Y 346.706,Z 447.733,A -85,B 0,C 180,E1 -13747.347,E2 -13747.347} C_VEL
LIN {X 0,Y 346.594,Z 450.024,A -85,B 0,C 180,E1 -13749.087,E2 -13749.087} C_VEL
LIN {X 0,Y 348.801,Z 460.14,A -85,B 0,C 180,E1 -13749.593,E2 -13749.593} C_VEL
LIN {X 0,Y 350.567,Z 469.496,A -85,B 0,C 180,E1 -13750.172,E2 -13750.172} C_VEL
LIN {X 0,Y 351.92,Z 478.671,A -85,B 0,C 180,E1 -13750.846,E2 -13750.846} C_VEL
LIN {X 0,Y 352.976,Z 487.116,A -85,B 0,C 180,E1 -13751.574,E2 -13751.574} C_VEL
LIN {X 0,Y 352.196,Z 496.399,A -85,B 0,C 180,E1 -13752.433,E2 -13752.433} C_VEL
LIN {X 0,Y 351.204,Z 505.346,A -85,B 0,C 180,E1 -13753.432,E2 -13753.432} C_VEL
LIN {X 0,Y 350.325,Z 513.526,A -85,B 0,C 180,E1 -13754.53,E2 -13754.53} C_VEL
LIN {X 0,Y 349.448,Z 521.104,A -85,B 0,C 180,E1 -13755.737,E2 -13755.737} C_VEL
LIN {X 0,Y 348.647,Z 527.307,A -85,B 0,C 180,E1 -13756.893,E2 -13756.893} C_VEL
LIN {X 0,Y 347.815,Z 533.846,A -85,B 0,C 180,E1 -13758.342,E2 -13758.342} C_VEL
LIN {X 0,Y 347.352,Z 538.352,A -85,B 0,C 180,E1 -13759.508,E2 -13759.508} C_VEL
LIN {X 0,Y 346.763,Z 543.846,A -85,B 0,C 180,E1 -13761.257,E2 -13761.257} C_VEL
LIN {X 0,Y 346.42,Z 548.175,A -85,B 0,C 180,E1 -13763.008,E2 -13763.008} C_VEL
LIN {X 0,Y 346.251,Z 550.543,A -85,B 0,C 180,E1 -13764.175,E2 -13764.175} C_VEL
LIN {X 0,Y 346.215,Z 552.345,A -85,B 0,C 180,E1 -13765.342,E2 -13765.342} C_VEL
LIN {X 0,Y 346.084,Z 554.791,A -85,B 0,C 180,E1 -13767.672,E2 -13767.672} C_VEL
LIN {X 0,Y 346.095,Z 555.38,A -85,B 0,C 180,E1 -13768.836,E2 -13768.836} C_VEL
LIN {X 0,Y 346.095,Z 555.381,A -85,B 0,C 180,E1 -13771.163,E2 -13771.163} C_VEL
LIN {X 0,Y 346.084,Z 554.791,A -85,B 0,C 180,E1 -13772.327,E2 -13772.327} C_VEL
LIN {X 0,Y 346.215,Z 552.345,A -85,B 0,C 180,E1 -13774.657,E2 -13774.657} C_VEL
LIN {X 0,Y 346.344,Z 549.395,A -85,B 0,C 180,E1 -13776.407,E2 -13776.407} C_VEL
LIN {X 0,Y 346.617,Z 545.402,A -85,B 0,C 180,E1 -13778.159,E2 -13778.159} C_VEL
LIN {X 0,Y 347.115,Z 540.27,A -85,B 0,C 180,E1 -13779.909,E2 -13779.909} C_VEL
LIN {X 0,Y 347.703,Z 535.005,A -85,B 0,C 180,E1 -13781.365,E2 -13781.365} C_VEL
LIN {X 0,Y 348.465,Z 528.686,A -85,B 0,C 180,E1 -13782.817,E2 -13782.817} C_VEL
LIN {X 0,Y 349.215,Z 522.734,A -85,B 0,C 180,E1 -13783.975,E2 -13783.975} C_VEL
LIN {X 0,Y 350.194,Z 514.682,A -85,B 0,C 180,E1 -13785.297,E2 -13785.297} C_VEL
LIN {X 0,Y 350.948,Z 507.621,A -85,B 0,C 180,E1 -13786.281,E2 -13786.281} C_VEL
LIN {X 0,Y 351.883,Z 499.107,A -85,B 0,C 180,E1 -13787.282,E2 -13787.282} C_VEL
LIN {X 0,Y 352.797,Z 490.39,A -85,B 0,C 180,E1 -13788.135,E2 -13788.135} C_VEL
LIN {X 0,Y 353.024,Z 487.123,A -85,B 0,C 180,E1 -13788.423,E2 -13788.423} C_VEL
LIN {X 0,Y 351.321,Z 473.72,A -85,B 0,C 180,E1 -13789.536,E2 -13789.536} C_VEL
LIN {X 0,Y 349.109,Z 461.553,A -85,B 0,C 180,E1 -13790.327,E2 -13790.327} C_VEL
LIN {X 0,Y 346.688,Z 450.876,A -85,B 0,C 180,E1 -13790.882,E2 -13790.882} C_VEL
LIN {X 0,Y 346.595,Z 449.96,A -85,B 0,C 180,E1 -13790.94,E2 -13790.94} C_VEL
LIN {X 0,Y 346.885,Z 445.612,A -85,B 0,C 180,E1 -13794.256,E2 -13794.256} C_VEL
LIN {X 0,Y 347.225,Z 441.131,A -85,B 0,C 180,E1 -13797.744,E2 -13797.744} C_VEL
LIN {X 0,Y 347.718,Z 436.221,A -85,B 0,C 180,E1 -13801.701,E2 -13801.701} C_VEL
LIN {X 0,Y 348.077,Z 432.99,A -85,B 0,C 180,E1 -13804.425,E2 -13804.425} C_VEL
LIN {X 0,Y 348.464,Z 429.787,A -85,B 0,C 180,E1 -13807.232,E2 -13807.232} C_VEL
LIN {X 0,Y 348.909,Z 426.646,A -85,B 0,C 180,E1 -13810.132,E2 -13810.132} C_VEL
LIN {X 0,Y 348.958,Z 423.538,A -85,B 0,C 180,E1 -13813.216,E2 -13813.216} C_VEL
LIN {X 0,Y 348.636,Z 420.478,A -85,B 0,C 180,E1 -13816.526,E2 -13816.526} C_VEL
LIN {X 0,Y 348.212,Z 417.519,A -85,B 0,C 180,E1 -13820.08,E2 -13820.08} C_VEL
LIN {X 0,Y 347.769,Z 414.669,A -85,B 0,C 180,E1 -13823.934,E2 -13823.934} C_VEL
LIN {X 0,Y 347.745,Z 414.671,A -85,B 0,C 180,E1 -13826.928,E2 -13826.928} C_VEL
LIN {X 0,Y 347.804,Z 414.663,A -85,B 0,C 180,E1 -13830.989,E2 -13830.989} C_VEL
LIN {X 0,Y 347.828,Z 414.655,A -85,B 0,C 180,E1 -13833.607,E2 -13833.607} C_VEL
LIN {X 0,Y 347.785,Z 414.662,A -85,B 0,C 180,E1 -13836.161,E2 -13836.161} C_VEL
LIN {X 0,Y 347.808,Z 414.658,A -85,B 0,C 180,E1 -13839.908,E2 -13839.908} C_VEL
LIN {X 0,Y 347.862,Z 414.654,A -85,B 0,C 180,E1 -13842.358,E2 -13842.358} C_VEL
LIN {X 0,Y 347.893,Z 414.647,A -85,B 0,C 180,E1 -13845.97,E2 -13845.97} C_VEL
LIN {X 0,Y 347.923,Z 414.643,A -85,B 0,C 180,E1 -13849.525,E2 -13849.525} C_VEL
LIN {X 0,Y 348.102,Z 414.622,A -85,B 0,C 180,E1 -13853.042,E2 -13853.042} C_VEL
LIN {X 0,Y 348.203,Z 414.608,A -85,B 0,C 180,E1 -13857.686,E2 -13857.686} C_VEL
LIN {X 0,Y 348.34,Z 414.593,A -85,B 0,C 180,E1 -13859.999,E2 -13859.999} C_VEL
LIN {X 0,Y 348.202,Z 414.612,A -85,B 0,C 180,E1 -13862.313,E2 -13862.313} C_VEL
LIN {X 0,Y 348.1,Z 414.621,A -85,B 0,C 180,E1 -13866.957,E2 -13866.957} C_VEL
LIN {X 0,Y 347.961,Z 414.638,A -85,B 0,C 180,E1 -13869.298,E2 -13869.298} C_VEL
LIN {X 0,Y 347.883,Z 414.649,A -85,B 0,C 180,E1 -13872.839,E2 -13872.839} C_VEL
LIN {X 0,Y 347.834,Z 414.657,A -85,B 0,C 180,E1 -13876.431,E2 -13876.431} C_VEL
LIN {X 0,Y 347.849,Z 414.652,A -85,B 0,C 180,E1 -13878.86,E2 -13878.86} C_VEL
LIN {X 0,Y 347.767,Z 414.664,A -85,B 0,C 180,E1 -13882.579,E2 -13882.579} C_VEL
LIN {X 0,Y 347.805,Z 414.657,A -85,B 0,C 180,E1 -13885.108,E2 -13885.108} C_VEL
LIN {X 0,Y 347.805,Z 414.661,A -85,B 0,C 180,E1 -13887.694,E2 -13887.694} C_VEL
LIN {X 0,Y 347.764,Z 414.665,A -85,B 0,C 180,E1 -13890.346,E2 -13890.346} C_VEL
LIN {X 0,Y 347.741,Z 414.67,A -85,B 0,C 180,E1 -13894.044,E2 -13894.044} C_VEL
LIN {X 0,Y 347.76,Z 414.665,A -85,B 0,C 180,E1 -13897.32,E2 -13897.32} C_VEL
LIN {X 0,Y 347.787,Z 414.661,A -85,B 0,C 180,E1 -13900.288,E2 -13900.288} C_VEL
LIN {X 0,Y 347.813,Z 414.659,A -85,B 0,C 180,E1 -13903.393,E2 -13903.393} C_VEL
LIN {X 0,Y 347.811,Z 414.657,A -85,B 0,C 180,E1 -13906.67,E2 -13906.67} C_VEL
LIN {X 0,Y 347.78,Z 414.662,A -85,B 0,C 180,E1 -13910.166,E2 -13910.166} C_VEL
LIN {X 0,Y 347.783,Z 414.661,A -85,B 0,C 180,E1 -13914.125,E2 -13914.125} C_VEL
LIN {X 0,Y 347.732,Z 414.668,A -85,B 0,C 180,E1 -13918.086,E2 -13918.086} C_VEL
LIN {X 0,Y 347.799,Z 414.66,A -85,B 0,C 180,E1 -13920.99,E2 -13920.99} C_VEL
LIN {X 0,Y 347.827,Z 414.659,A -85,B 0,C 180,E1 -13923.608,E2 -13923.608} C_VEL
LIN {X 0,Y 347.783,Z 414.661,A -85,B 0,C 180,E1 -13926.162,E2 -13926.162} C_VEL
LIN {X 0,Y 347.813,Z 414.661,A -85,B 0,C 180,E1 -13929.91,E2 -13929.91} C_VEL
LIN {X 0,Y 347.839,Z 414.658,A -85,B 0,C 180,E1 -13931.025,E2 -13931.025} C_VEL
LIN {X 0,Y 348.761,Z 417.376,A -85,B 0,C 180,E1 -13931.28,E2 -13931.28} C_VEL
LIN {X 0,Y 350.961,Z 419.676,A -85,B 0,C 180,E1 -13931.757,E2 -13931.757} C_VEL
LIN {X 0,Y 351.517,Z 420.252,A -85,B 0,C 180,E1 -13931.881,E2 -13931.881} C_VEL
LIN {X 0,Y 353.708,Z 423.583,A -85,B 0,C 180,E1 -13932.398,E2 -13932.398} C_VEL
LIN {X 0,Y 356.041,Z 425.863,A -85,B 0,C 180,E1 -13932.948,E2 -13932.948} C_VEL
LIN {X 0,Y 358.881,Z 429.481,A -85,B 0,C 180,E1 -13933.649,E2 -13933.649} C_VEL
LIN {X 0,Y 361.217,Z 431.648,A -85,B 0,C 180,E1 -13934.251,E2 -13934.251} C_VEL
LIN {X 0,Y 364.315,Z 435.291,A -85,B 0,C 180,E1 -13935.083,E2 -13935.083} C_VEL
LIN {X 0,Y 367.202,Z 437.842,A -85,B 0,C 180,E1 -13935.907,E2 -13935.907} C_VEL
LIN {X 0,Y 370.23,Z 441.274,A -85,B 0,C 180,E1 -13936.833,E2 -13936.833} C_VEL
LIN {X 0,Y 374.052,Z 444.353,A -85,B 0,C 180,E1 -13938.073,E2 -13938.073} C_VEL
LIN {X 0,Y 376.845,Z 447.451,A -85,B 0,C 180,E1 -13939.116,E2 -13939.116} C_VEL
LIN {X 0,Y 380.1,Z 449.912,A -85,B 0,C 180,E1 -13940.421,E2 -13940.421} C_VEL
LIN {X 0,Y 381.944,Z 451.005,A -85,B 0,C 180,E1 -13941.235,E2 -13941.235} C_VEL
LIN {X 0,Y 384.566,Z 454.124,A -85,B 0,C 180,E1 -13942.651,E2 -13942.651} C_VEL
LIN {X 0,Y 386.682,Z 455.953,A -85,B 0,C 180,E1 -13944.002,E2 -13944.002} C_VEL
LIN {X 0,Y 388.709,Z 457.143,A -85,B 0,C 180,E1 -13945.593,E2 -13945.593} C_VEL
LIN {X 0,Y 389.939,Z 457.474,A -85,B 0,C 180,E1 -13946.901,E2 -13946.901} C_VEL
LIN {X 0,Y 390.625,Z 457.632,A -85,B 0,C 180,E1 -13947.938,E2 -13947.938} C_VEL
LIN {X 0,Y 391.046,Z 457.676,A -85,B 0,C 180,E1 -13948.97,E2 -13948.97} C_VEL
LIN {X 0,Y 391.184,Z 457.719,A -85,B 0,C 180,E1 -13950,E2 -13950} C_VEL
LIN {X 0,Y 391.046,Z 457.679,A -85,B 0,C 180,E1 -13951.03,E2 -13951.03} C_VEL
LIN {X 0,Y 390.625,Z 457.62,A -85,B 0,C 180,E1 -13952.062,E2 -13952.062} C_VEL
LIN {X 0,Y 389.525,Z 457.37,A -85,B 0,C 180,E1 -13953.61,E2 -13953.61} C_VEL
LIN {X 0,Y 387.609,Z 456.543,A -85,B 0,C 180,E1 -13955.332,E2 -13955.332} C_VEL
LIN {X 0,Y 385.35,Z 454.9,A -85,B 0,C 180,E1 -13956.867,E2 -13956.867} C_VEL
LIN {X 0,Y 382.721,Z 452.042,A -85,B 0,C 180,E1 -13958.361,E2 -13958.361} C_VEL
LIN {X 0,Y 381.493,Z 450.58,A -85,B 0,C 180,E1 -13958.983,E2 -13958.983} C_VEL
LIN {X 0,Y 378.158,Z 448.585,A -85,B 0,C 180,E1 -13960.372,E2 -13960.372} C_VEL
LIN {X 0,Y 374.823,Z 445.372,A -85,B 0,C 180,E1 -13961.64,E2 -13961.64} C_VEL
LIN {X 0,Y 373.481,Z 443.681,A -85,B 0,C 180,E1 -13962.136,E2 -13962.136} C_VEL
LIN {X 0,Y 370.1,Z 441.159,A -85,B 0,C 180,E1 -13963.207,E2 -13963.207} C_VEL
LIN {X 0,Y 366.128,Z 436.763,A -85,B 0,C 180,E1 -13964.403,E2 -13964.403} C_VEL
LIN {X 0,Y 363.067,Z 434.02,A -85,B 0,C 180,E1 -13965.249,E2 -13965.249} C_VEL
LIN {X 0,Y 360.503,Z 430.835,A -85,B 0,C 180,E1 -13965.94,E2 -13965.94} C_VEL
LIN {X 0,Y 357.57,Z 428.075,A -85,B 0,C 180,E1 -13966.664,E2 -13966.664} C_VEL
LIN {X 0,Y 355.394,Z 425.099,A -85,B 0,C 180,E1 -13967.209,E2 -13967.209} C_VEL
LIN {X 0,Y 352.736,Z 422.383,A -85,B 0,C 180,E1 -13967.823,E2 -13967.823} C_VEL
LIN {X 0,Y 351.099,Z 419.764,A -85,B 0,C 180,E1 -13968.213,E2 -13968.213} C_VEL
LIN {X 0,Y 348.921,Z 417.617,A -85,B 0,C 180,E1 -13968.682,E2 -13968.682} C_VEL
LIN {X 0,Y 347.945,Z 415.329,A -85,B 0,C 180,E1 -13968.932,E2 -13968.932} C_VEL
LIN {X 0,Y 347.829,Z 414.66,A -85,B 0,C 180,E1 -13969.015,E2 -13969.015} C_VEL
LIN {X 0,Y 347.77,Z 414.668,A -85,B 0,C 180,E1 -13972.579,E2 -13972.579} C_VEL
LIN {X 0,Y 347.808,Z 414.659,A -85,B 0,C 180,E1 -13975.109,E2 -13975.109} C_VEL
LIN {X 0,Y 347.807,Z 414.658,A -85,B 0,C 180,E1 -13977.694,E2 -13977.694} C_VEL
LIN {X 0,Y 347.76,Z 414.668,A -85,B 0,C 180,E1 -13980.347,E2 -13980.347} C_VEL
LIN {X 0,Y 347.74,Z 414.672,A -85,B 0,C 180,E1 -13984.464,E2 -13984.464} C_VEL
LIN {X 0,Y 347.772,Z 414.664,A -85,B 0,C 180,E1 -13987.989,E2 -13987.989} C_VEL
LIN {X 0,Y 347.781,Z 414.662,A -85,B 0,C 180,E1 -13991.825,E2 -13991.825} C_VEL
LIN {X 0,Y 347.791,Z 414.66,A -85,B 0,C 180,E1 -13995.012,E2 -13995.012} C_VEL
LIN {X 0,Y 347.746,Z 414.669,A -85,B 0,C 180,E1 -13998.397,E2 -13998.397} C_VEL
LIN {X 0,Y 347.772,Z 414.666,A -85,B 0,C 180,E1 -14002.011,E2 -14002.011} C_VEL
LIN {X 0,Y 347.74,Z 414.667,A -85,B 0,C 180,E1 -14005.537,E2 -14005.537} C_VEL
LIN {X 0,Y 347.759,Z 414.665,A -85,B 0,C 180,E1 -14009.554,E2 -14009.554} C_VEL
LIN {X 0,Y 347.145,Z 414.746,A -85,B 0,C 180,E1 -14010.522,E2 -14010.522} C_VEL
LIN {X 0,Y 344.319,Z 415.1,A -85,B 0,C 180,E1 -14012.096,E2 -14012.096} C_VEL
LIN {X 0,Y 341.891,Z 415.399,A -85,B 0,C 180,E1 -14013.371,E2 -14013.371} C_VEL
LIN {X 0,Y 340.843,Z 415.527,A -85,B 0,C 180,E1 -14014.357,E2 -14014.357} C_VEL
LIN {X 0,Y 340.757,Z 415.535,A -85,B 0,C 180,E1 -14014.691,E2 -14014.691} C_VEL
LIN {X 0,Y 340.737,Z 415.541,A -85,B 0,C 180,E1 -14018.207,E2 -14018.207} C_VEL
LIN {X 0,Y 340.855,Z 415.529,A -85,B 0,C 180,E1 -14021.985,E2 -14021.985} C_VEL
LIN {X 0,Y 340.866,Z 415.526,A -85,B 0,C 180,E1 -14025.706,E2 -14025.706} C_VEL
LIN {X 0,Y 340.867,Z 415.523,A -85,B 0,C 180,E1 -14029.307,E2 -14029.307} C_VEL
LIN {X 0,Y 341.072,Z 415.497,A -85,B 0,C 180,E1 -14032.899,E2 -14032.899} C_VEL
LIN {X 0,Y 341.167,Z 415.487,A -85,B 0,C 180,E1 -14037.639,E2 -14037.639} C_VEL
LIN {X 0,Y 341.293,Z 415.47,A -85,B 0,C 180,E1 -14040.001,E2 -14040.001} C_VEL
LIN {X 0,Y 341.167,Z 415.485,A -85,B 0,C 180,E1 -14042.362,E2 -14042.362} C_VEL
LIN {X 0,Y 341.075,Z 415.498,A -85,B 0,C 180,E1 -14047.102,E2 -14047.102} C_VEL
LIN {X 0,Y 340.869,Z 415.522,A -85,B 0,C 180,E1 -14050.694,E2 -14050.694} C_VEL
LIN {X 0,Y 340.861,Z 415.523,A -85,B 0,C 180,E1 -14054.326,E2 -14054.326} C_VEL
LIN {X 0,Y 340.835,Z 415.526,A -85,B 0,C 180,E1 -14058.467,E2 -14058.467} C_VEL
LIN {X 0,Y 340.753,Z 415.537,A -85,B 0,C 180,E1 -14061.858,E2 -14061.858} C_VEL
LIN {X 0,Y 340.772,Z 415.536,A -85,B 0,C 180,E1 -14065.665,E2 -14065.665} C_VEL
LIN {X 0,Y 340.728,Z 415.54,A -85,B 0,C 180,E1 -14068.321,E2 -14068.321} C_VEL
LIN {X 0,Y 340.697,Z 415.549,A -85,B 0,C 180,E1 -14071.045,E2 -14071.045} C_VEL
LIN {X 0,Y 340.719,Z 415.546,A -85,B 0,C 180,E1 -14075.28,E2 -14075.28} C_VEL
LIN {X 0,Y 340.819,Z 416.245,A -85,B 0,C 180,E1 -14076.728,E2 -14076.728} C_VEL
LIN {X 0,Y 341.242,Z 418.968,A -85,B 0,C 180,E1 -14080.357,E2 -14080.357} C_VEL
LIN {X 0,Y 341.683,Z 422.354,A -85,B 0,C 180,E1 -14084.375,E2 -14084.375} C_VEL
LIN {X 0,Y 341.929,Z 425.032,A -85,B 0,C 180,E1 -14087.291,E2 -14087.291} C_VEL
LIN {X 0,Y 341.778,Z 428.141,A -85,B 0,C 180,E1 -14090.398,E2 -14090.398} C_VEL
LIN {X 0,Y 341.338,Z 431.379,A -85,B 0,C 180,E1 -14093.418,E2 -14093.418} C_VEL
LIN {X 0,Y 340.916,Z 434.487,A -85,B 0,C 180,E1 -14096.179,E2 -14096.179} C_VEL
LIN {X 0,Y 340.393,Z 439.143,A -85,B 0,C 180,E1 -14100.132,E2 -14100.132} C_VEL
LIN {X 0,Y 340.09,Z 442.622,A -85,B 0,C 180,E1 -14102.959,E2 -14102.959} C_VEL
LIN {X 0,Y 339.824,Z 445.903,A -85,B 0,C 180,E1 -14105.567,E2 -14105.567} C_VEL
LIN {X 0,Y 339.525,Z 449.795,A -85,B 0,C 180,E1 -14108.627,E2 -14108.627} C_VEL
LIN {X 0,Y 341.966,Z 460.716,A -85,B 0,C 180,E1 -14109.202,E2 -14109.202} C_VEL
LIN {X 0,Y 343.898,Z 471.142,A -85,B 0,C 180,E1 -14109.883,E2 -14109.883} C_VEL
LIN {X 0,Y 345.38,Z 481.938,A -85,B 0,C 180,E1 -14110.734,E2 -14110.734} C_VEL
LIN {X 0,Y 346.151,Z 488.539,A -85,B 0,C 180,E1 -14111.351,E2 -14111.351} C_VEL
LIN {X 0,Y 345.265,Z 497.539,A -85,B 0,C 180,E1 -14112.222,E2 -14112.222} C_VEL
LIN {X 0,Y 344.241,Z 506.269,A -85,B 0,C 180,E1 -14113.239,E2 -14113.239} C_VEL
LIN {X 0,Y 343.363,Z 514.093,A -85,B 0,C 180,E1 -14114.331,E2 -14114.331} C_VEL
LIN {X 0,Y 342.307,Z 522.519,A -85,B 0,C 180,E1 -14115.737,E2 -14115.737} C_VEL
LIN {X 0,Y 341.512,Z 528.471,A -85,B 0,C 180,E1 -14116.917,E2 -14116.917} C_VEL
LIN {X 0,Y 340.692,Z 534.79,A -85,B 0,C 180,E1 -14118.397,E2 -14118.397} C_VEL
LIN {X 0,Y 340.104,Z 540.056,A -85,B 0,C 180,E1 -14119.884,E2 -14119.884} C_VEL
LIN {X 0,Y 339.57,Z 545.189,A -85,B 0,C 180,E1 -14121.67,E2 -14121.67} C_VEL
LIN {X 0,Y 339.251,Z 549.18,A -85,B 0,C 180,E1 -14123.457,E2 -14123.457} C_VEL
LIN {X 0,Y 339.115,Z 552.133,A -85,B 0,C 180,E1 -14125.245,E2 -14125.245} C_VEL
LIN {X 0,Y 338.999,Z 554.58,A -85,B 0,C 180,E1 -14127.623,E2 -14127.623} C_VEL
LIN {X 0,Y 338.999,Z 555.169,A -85,B 0,C 180,E1 -14128.812,E2 -14128.812} C_VEL
LIN {X 0,Y 338.999,Z 555.169,A -85,B 0,C 180,E1 -14131.188,E2 -14131.188} C_VEL
LIN {X 0,Y 338.998,Z 554.58,A -85,B 0,C 180,E1 -14132.376,E2 -14132.376} C_VEL
LIN {X 0,Y 339.115,Z 552.133,A -85,B 0,C 180,E1 -14134.755,E2 -14134.755} C_VEL
LIN {X 0,Y 339.261,Z 549.182,A -85,B 0,C 180,E1 -14136.542,E2 -14136.542} C_VEL
LIN {X 0,Y 339.569,Z 545.19,A -85,B 0,C 180,E1 -14138.33,E2 -14138.33} C_VEL
LIN {X 0,Y 340.104,Z 540.058,A -85,B 0,C 180,E1 -14140.116,E2 -14140.116} C_VEL
LIN {X 0,Y 340.691,Z 534.792,A -85,B 0,C 180,E1 -14141.603,E2 -14141.603} C_VEL
LIN {X 0,Y 341.511,Z 528.474,A -85,B 0,C 180,E1 -14143.083,E2 -14143.083} C_VEL
LIN {X 0,Y 342.286,Z 522.521,A -85,B 0,C 180,E1 -14144.264,E2 -14144.264} C_VEL
LIN {X 0,Y 343.356,Z 514.122,A -85,B 0,C 180,E1 -14145.664,E2 -14145.664} C_VEL
LIN {X 0,Y 344.237,Z 506.273,A -85,B 0,C 180,E1 -14146.76,E2 -14146.76} C_VEL
LIN {X 0,Y 345.237,Z 497.543,A -85,B 0,C 180,E1 -14147.779,E2 -14147.779} C_VEL
LIN {X 0,Y 346.153,Z 488.545,A -85,B 0,C 180,E1 -14148.649,E2 -14148.649} C_VEL
LIN {X 0,Y 345.107,Z 479.209,A -85,B 0,C 180,E1 -14149.49,E2 -14149.49} C_VEL
LIN {X 0,Y 343.611,Z 469.214,A -85,B 0,C 180,E1 -14150.25,E2 -14150.25} C_VEL
LIN {X 0,Y 341.513,Z 458.557,A -85,B 0,C 180,E1 -14150.924,E2 -14150.924} C_VEL
LIN {X 0,Y 339.532,Z 449.771,A -85,B 0,C 180,E1 -14151.393,E2 -14151.393} C_VEL
LIN {X 0,Y 339.827,Z 445.82,A -85,B 0,C 180,E1 -14154.498,E2 -14154.498} C_VEL
LIN {X 0,Y 340.217,Z 440.995,A -85,B 0,C 180,E1 -14158.366,E2 -14158.366} C_VEL
LIN {X 0,Y 340.721,Z 436.095,A -85,B 0,C 180,E1 -14162.431,E2 -14162.431} C_VEL
LIN {X 0,Y 341.138,Z 432.878,A -85,B 0,C 180,E1 -14165.228,E2 -14165.228} C_VEL
LIN {X 0,Y 341.638,Z 429.211,A -85,B 0,C 180,E1 -14168.581,E2 -14168.581} C_VEL
LIN {X 0,Y 341.912,Z 426.575,A -85,B 0,C 180,E1 -14171.128,E2 -14171.128} C_VEL
LIN {X 0,Y 341.832,Z 423.488,A -85,B 0,C 180,E1 -14174.348,E2 -14174.348} C_VEL
LIN {X 0,Y 341.424,Z 420.458,A -85,B 0,C 180,E1 -14177.819,E2 -14177.819} C_VEL
LIN {X 0,Y 341.157,Z 418.454,A -85,B 0,C 180,E1 -14180.311,E2 -14180.311} C_VEL
LIN {X 0,Y 340.795,Z 416.055,A -85,B 0,C 180,E1 -14183.538,E2 -14183.538} C_VEL
LIN {X 0,Y 340.716,Z 415.547,A -85,B 0,C 180,E1 -14184.72,E2 -14184.72} C_VEL
LIN {X 0,Y 340.713,Z 415.547,A -85,B 0,C 180,E1 -14188.956,E2 -14188.956} C_VEL
LIN {X 0,Y 340.777,Z 415.536,A -85,B 0,C 180,E1 -14192.473,E2 -14192.473} C_VEL
LIN {X 0,Y 340.752,Z 415.537,A -85,B 0,C 180,E1 -14195.637,E2 -14195.637} C_VEL
LIN {X 0,Y 340.748,Z 415.538,A -85,B 0,C 180,E1 -14199.474,E2 -14199.474} C_VEL
LIN {X 0,Y 340.853,Z 415.525,A -85,B 0,C 180,E1 -14201.983,E2 -14201.983} C_VEL
LIN {X 0,Y 340.865,Z 415.522,A -85,B 0,C 180,E1 -14205.704,E2 -14205.704} C_VEL
LIN {X 0,Y 340.866,Z 415.522,A -85,B 0,C 180,E1 -14209.305,E2 -14209.305} C_VEL
LIN {X 0,Y 341.072,Z 415.499,A -85,B 0,C 180,E1 -14212.897,E2 -14212.897} C_VEL
LIN {X 0,Y 341.165,Z 415.485,A -85,B 0,C 180,E1 -14217.638,E2 -14217.638} C_VEL
LIN {X 0,Y 341.29,Z 415.471,A -85,B 0,C 180,E1 -14219.999,E2 -14219.999} C_VEL
LIN {X 0,Y 341.164,Z 415.487,A -85,B 0,C 180,E1 -14222.361,E2 -14222.361} C_VEL
LIN {X 0,Y 341.069,Z 415.497,A -85,B 0,C 180,E1 -14227.101,E2 -14227.101} C_VEL
LIN {X 0,Y 340.864,Z 415.524,A -85,B 0,C 180,E1 -14230.693,E2 -14230.693} C_VEL
LIN {X 0,Y 340.856,Z 415.527,A -85,B 0,C 180,E1 -14234.324,E2 -14234.324} C_VEL
LIN {X 0,Y 340.831,Z 415.529,A -85,B 0,C 180,E1 -14238.467,E2 -14238.467} C_VEL
LIN {X 0,Y 340.747,Z 415.541,A -85,B 0,C 180,E1 -14241.857,E2 -14241.857} C_VEL
LIN {X 0,Y 340.766,Z 415.536,A -85,B 0,C 180,E1 -14245.664,E2 -14245.664} C_VEL
LIN {X 0,Y 340.735,Z 415.541,A -85,B 0,C 180,E1 -14248.319,E2 -14248.319} C_VEL
LIN {X 0,Y 340.709,Z 415.542,A -85,B 0,C 180,E1 -14251.043,E2 -14251.043} C_VEL
LIN {X 0,Y 340.712,Z 415.542,A -85,B 0,C 180,E1 -14255.279,E2 -14255.279} C_VEL
LIN {X 0,Y 340.713,Z 415.542,A -85,B 0,C 180,E1 -14258.388,E2 -14258.388} C_VEL
LIN {X 0,Y 340.719,Z 415.542,A -85,B 0,C 180,E1 -14261.304,E2 -14261.304} C_VEL
LIN {X 0,Y 340.775,Z 415.534,A -85,B 0,C 180,E1 -14264.522,E2 -14264.522} C_VEL
LIN {X 0,Y 340.747,Z 415.54,A -85,B 0,C 180,E1 -14267.944,E2 -14267.944} C_VEL
LIN {X 0,Y 340.728,Z 415.54,A -85,B 0,C 180,E1 -14270.253,E2 -14270.253} C_VEL
LIN {X 0,Y 340.705,Z 415.548,A -85,B 0,C 180,E1 -14273.559,E2 -14273.559} C_VEL
LIN {X 0,Y 340.686,Z 415.545,A -85,B 0,C 180,E1 -14276.154,E2 -14276.154} C_VEL
LIN {X 0,Y 340.769,Z 415.535,A -85,B 0,C 180,E1 -14280.333,E2 -14280.333} C_VEL
LIN {X 0,Y 340.799,Z 415.533,A -85,B 0,C 180,E1 -14283.02,E2 -14283.02} C_VEL
LIN {X 0,Y 340.724,Z 415.543,A -85,B 0,C 180,E1 -14286.927,E2 -14286.927} C_VEL
LIN {X 0,Y 340.768,Z 415.539,A -85,B 0,C 180,E1 -14289.831,E2 -14289.831} C_VEL
LIN {X 0,Y 341.841,Z 418.506,A -85,B 0,C 180,E1 -14290.115,E2 -14290.115} C_VEL
LIN {X 0,Y 344.235,Z 421.121,A -85,B 0,C 180,E1 -14290.594,E2 -14290.594} C_VEL
LIN {X 0,Y 346.495,Z 424.413,A -85,B 0,C 180,E1 -14291.08,E2 -14291.08} C_VEL
LIN {X 0,Y 348.36,Z 426.344,A -85,B 0,C 180,E1 -14291.476,E2 -14291.476} C_VEL
LIN {X 0,Y 351.083,Z 429.952,A -85,B 0,C 180,E1 -14292.099,E2 -14292.099} C_VEL
LIN {X 0,Y 353.191,Z 432.043,A -85,B 0,C 180,E1 -14292.561,E2 -14292.561} C_VEL
LIN {X 0,Y 356.675,Z 436.109,A -85,B 0,C 180,E1 -14293.41,E2 -14293.41} C_VEL
LIN {X 0,Y 358.802,Z 438.11,A -85,B 0,C 180,E1 -14293.921,E2 -14293.921} C_VEL
LIN {X 0,Y 362.222,Z 441.875,A -85,B 0,C 180,E1 -14294.827,E2 -14294.827} C_VEL
LIN {X 0,Y 364.967,Z 444.321,A -85,B 0,C 180,E1 -14295.58,E2 -14295.58} C_VEL
LIN {X 0,Y 368.89,Z 448.391,A -85,B 0,C 180,E1 -14296.737,E2 -14296.737} C_VEL
LIN {X 0,Y 372.08,Z 450.857,A -85,B 0,C 180,E1 -14297.744,E2 -14297.744} C_VEL
LIN {X 0,Y 375.201,Z 454.171,A -85,B 0,C 180,E1 -14298.871,E2 -14298.871} C_VEL
LIN {X 0,Y 378.541,Z 456.644,A -85,B 0,C 180,E1 -14300.179,E2 -14300.179} C_VEL
LIN {X 0,Y 380.497,Z 457.878,A -85,B 0,C 180,E1 -14301.028,E2 -14301.028} C_VEL
LIN {X 0,Y 383.311,Z 461.132,A -85,B 0,C 180,E1 -14302.555,E2 -14302.555} C_VEL
LIN {X 0,Y 385.753,Z 463.131,A -85,B 0,C 180,E1 -14304.118,E2 -14304.118} C_VEL
LIN {X 0,Y 387.884,Z 464.26,A -85,B 0,C 180,E1 -14305.844,E2 -14305.844} C_VEL
LIN {X 0,Y 388.858,Z 464.484,A -85,B 0,C 180,E1 -14306.892,E2 -14306.892} C_VEL
LIN {X 0,Y 389.962,Z 464.692,A -85,B 0,C 180,E1 -14308.968,E2 -14308.968} C_VEL
LIN {X 0,Y 390.106,Z 464.736,A -85,B 0,C 180,E1 -14310,E2 -14310} C_VEL
LIN {X 0,Y 389.963,Z 464.673,A -85,B 0,C 180,E1 -14311.033,E2 -14311.033} C_VEL
LIN {X 0,Y 389.54,Z 464.635,A -85,B 0,C 180,E1 -14312.068,E2 -14312.068} C_VEL
LIN {X 0,Y 388.416,Z 464.366,A -85,B 0,C 180,E1 -14313.62,E2 -14313.62} C_VEL
LIN {X 0,Y 386.401,Z 463.514,A -85,B 0,C 180,E1 -14315.425,E2 -14315.425} C_VEL
LIN {X 0,Y 383.924,Z 461.709,A -85,B 0,C 180,E1 -14317.082,E2 -14317.082} C_VEL
LIN {X 0,Y 381.123,Z 458.699,A -85,B 0,C 180,E1 -14318.644,E2 -14318.644} C_VEL
LIN {X 0,Y 380.063,Z 457.448,A -85,B 0,C 180,E1 -14319.168,E2 -14319.168} C_VEL
LIN {X 0,Y 376.595,Z 455.35,A -85,B 0,C 180,E1 -14320.597,E2 -14320.597} C_VEL
LIN {X 0,Y 373.025,Z 451.987,A -85,B 0,C 180,E1 -14321.925,E2 -14321.925} C_VEL
LIN {X 0,Y 371.175,Z 450.061,A -85,B 0,C 180,E1 -14322.554,E2 -14322.554} C_VEL
LIN {X 0,Y 367.545,Z 447.145,A -85,B 0,C 180,E1 -14323.67,E2 -14323.67} C_VEL
LIN {X 0,Y 363.849,Z 443.156,A -85,B 0,C 180,E1 -14324.749,E2 -14324.749} C_VEL
LIN {X 0,Y 360.112,Z 439.806,A -85,B 0,C 180,E1 -14325.721,E2 -14325.721} C_VEL
LIN {X 0,Y 357.641,Z 436.884,A -85,B 0,C 180,E1 -14326.368,E2 -14326.368} C_VEL
LIN {X 0,Y 354.116,Z 433.331,A -85,B 0,C 180,E1 -14327.209,E2 -14327.209} C_VEL
LIN {X 0,Y 352.211,Z 430.967,A -85,B 0,C 180,E1 -14327.658,E2 -14327.658} C_VEL
LIN {X 0,Y 349.103,Z 427.557,A -85,B 0,C 180,E1 -14328.35,E2 -14328.35} C_VEL
LIN {X 0,Y 347.585,Z 425.434,A -85,B 0,C 180,E1 -14328.694,E2 -14328.694} C_VEL
LIN {X 0,Y 345.115,Z 422.671,A -85,B 0,C 180,E1 -14329.211,E2 -14329.211} C_VEL
LIN {X 0,Y 343.719,Z 420.46,A -85,B 0,C 180,E1 -14329.512,E2 -14329.512} C_VEL
LIN {X 0,Y 341.672,Z 418.202,A -85,B 0,C 180,E1 -14329.922,E2 -14329.922} C_VEL
LIN {X 0,Y 340.773,Z 415.538,A -85,B 0,C 180,E1 -14330.188,E2 -14330.188} C_VEL
LIN {X 0,Y 340.725,Z 415.542,A -85,B 0,C 180,E1 -14333.073,E2 -14333.073} C_VEL
LIN {X 0,Y 340.801,Z 415.533,A -85,B 0,C 180,E1 -14336.98,E2 -14336.98} C_VEL
LIN {X 0,Y 340.759,Z 415.537,A -85,B 0,C 180,E1 -14339.978,E2 -14339.978} C_VEL
LIN {X 0,Y 340.688,Z 415.545,A -85,B 0,C 180,E1 -14343.847,E2 -14343.847} C_VEL
LIN {X 0,Y 340.702,Z 415.546,A -85,B 0,C 180,E1 -14346.742,E2 -14346.742} C_VEL
LIN {X 0,Y 340.76,Z 415.54,A -85,B 0,C 180,E1 -14350.262,E2 -14350.262} C_VEL
LIN {X 0,Y 340.713,Z 415.542,A -85,B 0,C 180,E1 -14353.785,E2 -14353.785} C_VEL
LIN {X 0,Y 340.674,Z 415.546,A -85,B 0,C 180,E1 -14357.096,E2 -14357.096} C_VEL
LIN {X 0,Y 340.695,Z 415.549,A -85,B 0,C 180,E1 -14360.248,E2 -14360.248} C_VEL
LIN {X 0,Y 340.707,Z 415.543,A -85,B 0,C 180,E1 -14363.559,E2 -14363.559} C_VEL
LIN {X 0,Y 340.691,Z 415.55,A -85,B 0,C 180,E1 -14366.154,E2 -14366.154} C_VEL
LIN {X 0,Y 340.771,Z 415.537,A -85,B 0,C 180,E1 -14370.333,E2 -14370.333} C_VEL
LIN {X 0,Y 340.801,Z 415.53,A -85,B 0,C 180,E1 -14373.021,E2 -14373.021} C_VEL
LIN {X 0,Y 340.757,Z 415.535,A -85,B 0,C 180,E1 -14374.691,E2 -14374.691} C_VEL
LIN {X 0,Y 340.075,Z 415.625,A -85,B 0,C 180,E1 -14375.678,E2 -14375.678} C_VEL
LIN {X 0,Y 337.18,Z 415.982,A -85,B 0,C 180,E1 -14377.283,E2 -14377.283} C_VEL
LIN {X 0,Y 334.759,Z 416.283,A -85,B 0,C 180,E1 -14378.583,E2 -14378.583} C_VEL
LIN {X 0,Y 333.761,Z 416.409,A -85,B 0,C 180,E1 -14379.589,E2 -14379.589} C_VEL
LIN {X 0,Y 333.701,Z 416.414,A -85,B 0,C 180,E1 -14379.93,E2 -14379.93} C_VEL
LIN {X 0,Y 333.744,Z 416.409,A -85,B 0,C 180,E1 -14382.854,E2 -14382.854} C_VEL
LIN {X 0,Y 333.793,Z 416.403,A -85,B 0,C 180,E1 -14386.609,E2 -14386.609} C_VEL
LIN {X 0,Y 333.859,Z 416.395,A -85,B 0,C 180,E1 -14390.306,E2 -14390.306} C_VEL
LIN {X 0,Y 334.022,Z 416.375,A -85,B 0,C 180,E1 -14392.748,E2 -14392.748} C_VEL
LIN {X 0,Y 333.808,Z 416.402,A -85,B 0,C 180,E1 -14395.17,E2 -14395.17} C_VEL
LIN {X 0,Y 334.104,Z 416.366,A -85,B 0,C 180,E1 -14397.589,E2 -14397.589} C_VEL
LIN {X 0,Y 334.244,Z 416.348,A -85,B 0,C 180,E1 -14400.001,E2 -14400.001} C_VEL
LIN {X 0,Y 334.105,Z 416.364,A -85,B 0,C 180,E1 -14402.412,E2 -14402.412} C_VEL
LIN {X 0,Y 334.024,Z 416.378,A -85,B 0,C 180,E1 -14407.253,E2 -14407.253} C_VEL
LIN {X 0,Y 333.832,Z 416.4,A -85,B 0,C 180,E1 -14410.923,E2 -14410.923} C_VEL
LIN {X 0,Y 333.807,Z 416.402,A -85,B 0,C 180,E1 -14414.635,E2 -14414.635} C_VEL
LIN {X 0,Y 333.794,Z 416.404,A -85,B 0,C 180,E1 -14418.655,E2 -14418.655} C_VEL
LIN {X 0,Y 333.691,Z 416.416,A -85,B 0,C 180,E1 -14422.279,E2 -14422.279} C_VEL
LIN {X 0,Y 333.734,Z 416.411,A -85,B 0,C 180,E1 -14426.247,E2 -14426.247} C_VEL
LIN {X 0,Y 333.689,Z 416.421,A -85,B 0,C 180,E1 -14428.975,E2 -14428.975} C_VEL
LIN {X 0,Y 333.643,Z 416.425,A -85,B 0,C 180,E1 -14432.588,E2 -14432.588} C_VEL
LIN {X 0,Y 333.686,Z 416.422,A -85,B 0,C 180,E1 -14434.775,E2 -14434.775} C_VEL
LIN {X 0,Y 333.818,Z 417.49,A -85,B 0,C 180,E1 -14436.868,E2 -14436.868} C_VEL
LIN {X 0,Y 334.281,Z 420.438,A -85,B 0,C 180,E1 -14440.811,E2 -14440.811} C_VEL
LIN {X 0,Y 334.678,Z 423.435,A -85,B 0,C 180,E1 -14444.441,E2 -14444.441} C_VEL
LIN {X 0,Y 334.902,Z 426.506,A -85,B 0,C 180,E1 -14447.815,E2 -14447.815} C_VEL
LIN {X 0,Y 334.836,Z 428.063,A -85,B 0,C 180,E1 -14449.408,E2 -14449.408} C_VEL
LIN {X 0,Y 334.352,Z 431.798,A -85,B 0,C 180,E1 -14453.012,E2 -14453.012} C_VEL
LIN {X 0,Y 333.758,Z 435.975,A -85,B 0,C 180,E1 -14456.805,E2 -14456.805} C_VEL
LIN {X 0,Y 333.217,Z 440.827,A -85,B 0,C 180,E1 -14460.981,E2 -14460.981} C_VEL
LIN {X 0,Y 332.887,Z 444.082,A -85,B 0,C 180,E1 -14463.682,E2 -14463.682} C_VEL
LIN {X 0,Y 332.629,Z 447.378,A -85,B 0,C 180,E1 -14466.332,E2 -14466.332} C_VEL
LIN {X 0,Y 332.473,Z 449.695,A -85,B 0,C 180,E1 -14468.158,E2 -14468.158} C_VEL
LIN {X 0,Y 334.711,Z 459.302,A -85,B 0,C 180,E1 -14468.675,E2 -14468.675} C_VEL
LIN {X 0,Y 336.602,Z 469.071,A -85,B 0,C 180,E1 -14469.314,E2 -14469.314} C_VEL
LIN {X 0,Y 338.118,Z 479.044,A -85,B 0,C 180,E1 -14470.095,E2 -14470.095} C_VEL
LIN {X 0,Y 339.203,Z 488.32,A -85,B 0,C 180,E1 -14470.954,E2 -14470.954} C_VEL
LIN {X 0,Y 338.816,Z 494.624,A -85,B 0,C 180,E1 -14471.559,E2 -14471.559} C_VEL
LIN {X 0,Y 337.548,Z 504.922,A -85,B 0,C 180,E1 -14472.741,E2 -14472.741} C_VEL
LIN {X 0,Y 336.544,Z 513.028,A -85,B 0,C 180,E1 -14473.867,E2 -14473.867} C_VEL
LIN {X 0,Y 335.607,Z 520.678,A -85,B 0,C 180,E1 -14475.136,E2 -14475.136} C_VEL
LIN {X 0,Y 334.783,Z 526.883,A -85,B 0,C 180,E1 -14476.339,E2 -14476.339} C_VEL
LIN {X 0,Y 333.862,Z 533.422,A -85,B 0,C 180,E1 -14477.848,E2 -14477.848} C_VEL
LIN {X 0,Y 333.353,Z 537.928,A -85,B 0,C 180,E1 -14479.062,E2 -14479.062} C_VEL
LIN {X 0,Y 332.678,Z 543.422,A -85,B 0,C 180,E1 -14480.883,E2 -14480.883} C_VEL
LIN {X 0,Y 332.28,Z 547.751,A -85,B 0,C 180,E1 -14482.709,E2 -14482.709} C_VEL
LIN {X 0,Y 332.074,Z 550.387,A -85,B 0,C 180,E1 -14484.106,E2 -14484.106} C_VEL
LIN {X 0,Y 332.005,Z 553.311,A -85,B 0,C 180,E1 -14486.359,E2 -14486.359} C_VEL
LIN {X 0,Y 331.916,Z 554.369,A -85,B 0,C 180,E1 -14487.573,E2 -14487.573} C_VEL
LIN {X 0,Y 331.905,Z 554.958,A -85,B 0,C 180,E1 -14488.786,E2 -14488.786} C_VEL
LIN {X 0,Y 331.905,Z 554.958,A -85,B 0,C 180,E1 -14491.213,E2 -14491.213} C_VEL
LIN {X 0,Y 331.916,Z 554.369,A -85,B 0,C 180,E1 -14492.427,E2 -14492.427} C_VEL
LIN {X 0,Y 332.021,Z 551.922,A -85,B 0,C 180,E1 -14494.857,E2 -14494.857} C_VEL
LIN {X 0,Y 332.185,Z 548.97,A -85,B 0,C 180,E1 -14496.682,E2 -14496.682} C_VEL
LIN {X 0,Y 332.513,Z 544.978,A -85,B 0,C 180,E1 -14498.508,E2 -14498.508} C_VEL
LIN {X 0,Y 333.086,Z 539.846,A -85,B 0,C 180,E1 -14500.331,E2 -14500.331} C_VEL
LIN {X 0,Y 333.705,Z 534.58,A -85,B 0,C 180,E1 -14501.849,E2 -14501.849} C_VEL
LIN {X 0,Y 334.571,Z 528.262,A -85,B 0,C 180,E1 -14503.359,E2 -14503.359} C_VEL
LIN {X 0,Y 335.364,Z 522.308,A -85,B 0,C 180,E1 -14504.564,E2 -14504.564} C_VEL
LIN {X 0,Y 336.392,Z 514.716,A -85,B 0,C 180,E1 -14505.867,E2 -14505.867} C_VEL
LIN {X 0,Y 337.413,Z 506.061,A -85,B 0,C 180,E1 -14507.11,E2 -14507.11} C_VEL
LIN {X 0,Y 338.455,Z 497.331,A -85,B 0,C 180,E1 -14508.148,E2 -14508.148} C_VEL
LIN {X 0,Y 339.28,Z 489.966,A -85,B 0,C 180,E1 -14508.884,E2 -14508.884} C_VEL
LIN {X 0,Y 338.403,Z 481.044,A -85,B 0,C 180,E1 -14509.732,E2 -14509.732} C_VEL
LIN {X 0,Y 336.97,Z 470.912,A -85,B 0,C 180,E1 -14510.55,E2 -14510.55} C_VEL
LIN {X 0,Y 334.959,Z 460.406,A -85,B 0,C 180,E1 -14511.258,E2 -14511.258} C_VEL
LIN {X 0,Y 332.472,Z 449.56,A -85,B 0,C 180,E1 -14511.885,E2 -14511.885} C_VEL
LIN {X 0,Y 332.773,Z 445.739,A -85,B 0,C 180,E1 -14514.985,E2 -14514.985} C_VEL
LIN {X 0,Y 333.068,Z 442.454,A -85,B 0,C 180,E1 -14517.659,E2 -14517.659} C_VEL
LIN {X 0,Y 333.547,Z 437.575,A -85,B 0,C 180,E1 -14521.786,E2 -14521.786} C_VEL
LIN {X 0,Y 334.031,Z 434.102,A -85,B 0,C 180,E1 -14524.858,E2 -14524.858} C_VEL
LIN {X 0,Y 334.402,Z 431.193,A -85,B 0,C 180,E1 -14527.551,E2 -14527.551} C_VEL
LIN {X 0,Y 334.857,Z 427.724,A -85,B 0,C 180,E1 -14530.924,E2 -14530.924} C_VEL
LIN {X 0,Y 334.836,Z 424.96,A -85,B 0,C 180,E1 -14533.839,E2 -14533.839} C_VEL
LIN {X 0,Y 334.459,Z 421.925,A -85,B 0,C 180,E1 -14537.344,E2 -14537.344} C_VEL
LIN {X 0,Y 334.06,Z 419.122,A -85,B 0,C 180,E1 -14540.865,E2 -14540.865} C_VEL
LIN {X 0,Y 333.758,Z 416.972,A -85,B 0,C 180,E1 -14543.871,E2 -14543.871} C_VEL
LIN {X 0,Y 333.672,Z 416.424,A -85,B 0,C 180,E1 -14545.34,E2 -14545.34} C_VEL
LIN {X 0,Y 333.697,Z 416.416,A -85,B 0,C 180,E1 -14549.637,E2 -14549.637} C_VEL
LIN {X 0,Y 333.741,Z 416.412,A -85,B 0,C 180,E1 -14552.4,E2 -14552.4} C_VEL
LIN {X 0,Y 333.723,Z 416.416,A -85,B 0,C 180,E1 -14555.09,E2 -14555.09} C_VEL
LIN {X 0,Y 333.681,Z 416.421,A -85,B 0,C 180,E1 -14559.019,E2 -14559.019} C_VEL
LIN {X 0,Y 333.789,Z 416.404,A -85,B 0,C 180,E1 -14561.589,E2 -14561.589} C_VEL
LIN {X 0,Y 333.804,Z 416.402,A -85,B 0,C 180,E1 -14565.576,E2 -14565.576} C_VEL
LIN {X 0,Y 333.829,Z 416.4,A -85,B 0,C 180,E1 -14569.077,E2 -14569.077} C_VEL
LIN {X 0,Y 334.021,Z 416.378,A -85,B 0,C 180,E1 -14572.747,E2 -14572.747} C_VEL
LIN {X 0,Y 333.807,Z 416.402,A -85,B 0,C 180,E1 -14575.168,E2 -14575.168} C_VEL
LIN {X 0,Y 334.102,Z 416.365,A -85,B 0,C 180,E1 -14577.588,E2 -14577.588} C_VEL
LIN {X 0,Y 334.241,Z 416.348,A -85,B 0,C 180,E1 -14579.999,E2 -14579.999} C_VEL
LIN {X 0,Y 334.102,Z 416.366,A -85,B 0,C 180,E1 -14582.411,E2 -14582.411} C_VEL
LIN {X 0,Y 334.019,Z 416.375,A -85,B 0,C 180,E1 -14587.252,E2 -14587.252} C_VEL
LIN {X 0,Y 333.827,Z 416.399,A -85,B 0,C 180,E1 -14590.921,E2 -14590.921} C_VEL
LIN {X 0,Y 333.802,Z 416.403,A -85,B 0,C 180,E1 -14594.634,E2 -14594.634} C_VEL
LIN {X 0,Y 333.79,Z 416.404,A -85,B 0,C 180,E1 -14598.655,E2 -14598.655} C_VEL
LIN {X 0,Y 333.686,Z 416.42,A -85,B 0,C 180,E1 -14602.278,E2 -14602.278} C_VEL
LIN {X 0,Y 333.729,Z 416.414,A -85,B 0,C 180,E1 -14606.246,E2 -14606.246} C_VEL
LIN {X 0,Y 333.705,Z 416.414,A -85,B 0,C 180,E1 -14608.972,E2 -14608.972} C_VEL
LIN {X 0,Y 333.645,Z 416.422,A -85,B 0,C 180,E1 -14612.589,E2 -14612.589} C_VEL
LIN {X 0,Y 333.671,Z 416.421,A -85,B 0,C 180,E1 -14616.139,E2 -14616.139} C_VEL
LIN {X 0,Y 333.678,Z 416.418,A -85,B 0,C 180,E1 -14619.187,E2 -14619.187} C_VEL
LIN {X 0,Y 333.697,Z 416.415,A -85,B 0,C 180,E1 -14622.513,E2 -14622.513} C_VEL
LIN {X 0,Y 333.723,Z 416.415,A -85,B 0,C 180,E1 -14625.977,E2 -14625.977} C_VEL
LIN {X 0,Y 333.696,Z 416.418,A -85,B 0,C 180,E1 -14629.305,E2 -14629.305} C_VEL
LIN {X 0,Y 333.66,Z 416.422,A -85,B 0,C 180,E1 -14633.168,E2 -14633.168} C_VEL
LIN {X 0,Y 333.668,Z 416.423,A -85,B 0,C 180,E1 -14635.342,E2 -14635.342} C_VEL
LIN {X 0,Y 333.697,Z 416.419,A -85,B 0,C 180,E1 -14639.71,E2 -14639.71} C_VEL
LIN {X 0,Y 333.738,Z 416.411,A -85,B 0,C 180,E1 -14642.401,E2 -14642.401} C_VEL
LIN {X 0,Y 333.722,Z 416.416,A -85,B 0,C 180,E1 -14645.091,E2 -14645.091} C_VEL
LIN {X 0,Y 333.704,Z 416.479,A -85,B 0,C 180,E1 -14648.78,E2 -14648.78} C_VEL
LIN {X 0,Y 334.702,Z 419.297,A -85,B 0,C 180,E1 -14649.01,E2 -14649.01} C_VEL
LIN {X 0,Y 336.956,Z 421.984,A -85,B 0,C 180,E1 -14649.431,E2 -14649.431} C_VEL
LIN {X 0,Y 339.21,Z 425.264,A -85,B 0,C 180,E1 -14649.878,E2 -14649.878} C_VEL
LIN {X 0,Y 340.839,Z 427.193,A -85,B 0,C 180,E1 -14650.199,E2 -14650.199} C_VEL
LIN {X 0,Y 343.893,Z 430.924,A -85,B 0,C 180,E1 -14650.82,E2 -14650.82} C_VEL
LIN {X 0,Y 348.628,Z 436.472,A -85,B 0,C 180,E1 -14651.834,E2 -14651.834} C_VEL
LIN {X 0,Y 353.799,Z 442.125,A -85,B 0,C 180,E1 -14653.01,E2 -14653.01} C_VEL
LIN {X 0,Y 356.586,Z 444.89,A -85,B 0,C 180,E1 -14653.673,E2 -14653.673} C_VEL
LIN {X 0,Y 359.958,Z 448.363,A -85,B 0,C 180,E1 -14654.539,E2 -14654.539} C_VEL
LIN {X 0,Y 362.712,Z 450.799,A -85,B 0,C 180,E1 -14655.268,E2 -14655.268} C_VEL
LIN {X 0,Y 366.871,Z 455.028,A -85,B 0,C 180,E1 -14656.497,E2 -14656.497} C_VEL
LIN {X 0,Y 370.235,Z 457.747,A -85,B 0,C 180,E1 -14657.564,E2 -14657.564} C_VEL
LIN {X 0,Y 373.473,Z 461.102,A -85,B 0,C 180,E1 -14658.759,E2 -14658.759} C_VEL
LIN {X 0,Y 377.294,Z 463.788,A -85,B 0,C 180,E1 -14660.248,E2 -14660.248} C_VEL
LIN {X 0,Y 378.654,Z 464.644,A -85,B 0,C 180,E1 -14660.836,E2 -14660.836} C_VEL
LIN {X 0,Y 381.453,Z 467.865,A -85,B 0,C 180,E1 -14662.376,E2 -14662.376} C_VEL
LIN {X 0,Y 383.848,Z 469.829,A -85,B 0,C 180,E1 -14663.891,E2 -14663.891} C_VEL
LIN {X 0,Y 386.041,Z 471.072,A -85,B 0,C 180,E1 -14665.615,E2 -14665.615} C_VEL
LIN {X 0,Y 387.269,Z 471.404,A -85,B 0,C 180,E1 -14666.879,E2 -14666.879} C_VEL
LIN {X 0,Y 387.975,Z 471.572,A -85,B 0,C 180,E1 -14667.924,E2 -14667.924} C_VEL
LIN {X 0,Y 388.423,Z 471.623,A -85,B 0,C 180,E1 -14668.963,E2 -14668.963} C_VEL
LIN {X 0,Y 388.571,Z 471.667,A -85,B 0,C 180,E1 -14670,E2 -14670} C_VEL
LIN {X 0,Y 388.419,Z 471.598,A -85,B 0,C 180,E1 -14671.037,E2 -14671.037} C_VEL
LIN {X 0,Y 387.275,Z 471.375,A -85,B 0,C 180,E1 -14673.121,E2 -14673.121} C_VEL
LIN {X 0,Y 385.349,Z 470.737,A -85,B 0,C 180,E1 -14674.979,E2 -14674.979} C_VEL
